FUNCTION "Axis_Control" : VOID	// FC 38
TITLE = Axis control
//KNOW_HOW_PROTECT
//
VERSION : 0.1
VAR_INPUT
  Enable : BOOL ;
  Axis_Enc_Num : BYTE ;
  Axis_Plus_LimitSwitch : BOOL ;
  Axis_Minus_LimitSwitch : BOOL ;
  Axis_Ref_Switch : BOOL ;
  Axis_PositContr : BOOL ;
  Run_Mode : BOOL ;
  Axis_1st_Ref_Active : BOOL ;
  Axis_2nd_Ref_Active : BOOL ;
  Axis_Limitactive : DWORD ;
END_VAR
VAR_OUTPUT
  Axis_PulseEnable : BOOL ;
  Axis_ContrEnable : BOOL ;
  Axis_PosMeas1 : BOOL ;
  Axis_PosMeas2 : BOOL ;
  Axis_ORactive : BOOL ;
  Axis_Refactive : BOOL ;
  Axis_BreakActive : BOOL ;
  Axis_Plus_Limit : BOOL ;
  Axis_Minus_Limit : BOOL ;
  Axis_refpoint : BOOL ;
END_VAR
BEGIN
NETWORK
TITLE =
      L     1;
      L     #Axis_Enc_Num;
      -I;
      JN    M001;
      A     "ONE";
      =     #Axis_PosMeas1;
      AN    #Axis_PosMeas1;
      =     #Axis_PosMeas2;
      JU    M002;
M001: A     "ONE";
      =     #Axis_PosMeas2;
      AN    #Axis_PosMeas2;
      =     #Axis_PosMeas1;
M002: A     #Enable;
      =     #Axis_PulseEnable;
      =     #Axis_ContrEnable;
      AN    #Run_Mode;
      =     #Axis_ORactive;
      A     #Axis_PositContr;
      =     #Axis_BreakActive;
      A     #Axis_1st_Ref_Active;
      O     #Axis_2nd_Ref_Active;
      =     #Axis_Refactive;
      A     #Axis_Ref_Switch;
      =     #Axis_refpoint;
      L     #Axis_Limitactive;
      L     1.000000e+00;
      -R;
      JZ    NONE;
      AN    #Axis_Plus_LimitSwitch;
      =     #Axis_Plus_Limit;
      AN    #Axis_Minus_LimitSwitch;
      =     #Axis_Minus_Limit;
      JU    EXIT;
NONE: A     "Reset_Key";
      R     #Axis_Plus_Limit;
      R     #Axis_Minus_Limit;
EXIT: BE;
END_FUNCTION

FUNCTION "System_Date" : VOID	// FC 39
TITLE = function
//KNOW_HOW_PROTECT 
//M153.6,MW316 DB110,DB120,DB125
//
VERSION : 0.1
BEGIN
NETWORK
TITLE =
//ReadSysTime M153.6,MW316 DB110,DB120,DB125
      CALL  "READ_CLK" (
           RET_VAL                  := MW 316,
           CDT                      := P#DB110.DBX 0.0);
      L     DB110.DBB 0;	//YEAR
      BTI;
      T     DB125.DBB 0;
      T     "USER_DB5".STAT0[5];
      L     DB110.DBB 1;	//MONTH
      BTI;
      T     DB125.DBB 1;
      T     "USER_DB5".STAT0[6];
      L     DB110.DBB 2;	//DAY
      BTI;
      T     DB125.DBB 2;
      T     "USER_DB5".STAT0[7];
      L     DB110.DBB 3;	//HOUR
      BTI;
      T     DB125.DBB 3;
      T     "USER_DB5".STAT0[8];
      L     DB110.DBB 4;	//MINUTE
      BTI;
      T     DB125.DBB 4;
      T     "USER_DB5".STAT0[9];
      L     DB110.DBB 5;	//SECOND
      BTI;
      T     DB125.DBB 5;
      T     "USER_DB5".STAT0[10];
      A     "Time_Lock_Active";
      JC    EXIT;
      L     DB120.DBD 70;
      L     1.000000e+00;
      -R;
      JN    ZERO;
      L     "USER_DB5".STAT0[5];	//YEAR
      L     10000;
      *I;
      T     DB125.DBD 30;
      L     "USER_DB5".STAT0[6];	//MONTH
      L     100;
      *I;
      T     DB125.DBD 40;
      L     "USER_DB5".STAT0[7];	//DATE
      T     DB125.DBD 50;
      L     DB125.DBD 30;
      +D;
      T     DB125.DBD 60;
      L     DB125.DBD 40;
      +D;
      T     DB125.DBD 70;
      L     DB120.DBD 80;
      RND;
      T     DB125.DBD 80;
      L     DB125.DBD 70;
      L     DB125.DBD 80;
      >=I;
      JC    ONE;
      JU    ZERO;
EXIT: L     DB120.DBD 70;
      L     1.000000e+00;
      -R;
      JZ    ONE;
      A     "Reset_Key";
      A     "Auto_Key";
      A     "MDA_Key";
      R     "Time_Lock_Active";
      JU    END;
ONE:  S     "Time_Lock_Active";
      JU    END;
ZERO: R     "Time_Lock_Active";
END:  BE;
END_FUNCTION

FUNCTION "X_BACK_Control" : VOID	// FC 40
TITLE = X_BACK
//M155.0_M155.7,MW322,MW324,DB16,DB106,DB159,FB4,FC9,T27
//KNOW_HOW_PROTECT
//
VERSION : 0.1
BEGIN
NETWORK
TITLE = M155.0_M155.7,MW322,MW324,DB16,DB106,DB159,FB4,FC9,T27
      A     "Auto_LED";
      L     S5T#500MS;
      SD    "KT17";
      A     "KT17";
      =     M 155.0;
      A     "Reset_Key";
      A     M 155.1;
      R     M 155.0;
      R     M 155.1;
      CALL  "PI_SERV" , DB 159 (
           DIX 0.0                  := M 155.0,
           DIW 2                    := W#16#1002,
           DIW 4                    := 26,
           DIW 6                    := 16,
           DID 8                    := P#DBX 18.0,
           DIW 12                   := 1,
           DIW 14                   := W#16#1002,
           DIW 16                   := 34,
           DIW 18                   := 106,
           DID 20                   := P#DBX 34.0,
           DIW 24                   := W#16#1002,
           DIW 26                   := 34,
           DIW 28                   := 106,
           DID 30                   := P#DBX 0.0,
           DIW 54                   := 1,
           DIW 56                   := 1,
           DIX 74.0                 := M 155.1,
           DIX 74.1                 := M 155.2,
           DIW 76                   := MW 322);
      A(;
      O     DB11.DBX 6.0;
      O     DB11.DBX 6.1;
      );
      A     DB21.DBX 35.0;
      AN    DB21.DBX 197.6;
      AN    "Reset_Key";
      =     M 156.0;
      CALL  "Single Key control" (
           CH1_M_ON                 := DB21.DBX 201.0,
           CH2_M_ON                 := FALSE,
           CH1_M_OFF                := DB21.DBX 201.1,
           CH2_M_OFF                := FALSE,
           Key                      := "T13_X轴快退",
           Var1                     := M 156.1,
           Var2                     := M 156.2,
           Var3_up                  := FALSE,
           Protect                  := M 156.0,
           KeyEnableMode            := TRUE,
           KA                       := M 156.3,
           LED                      := M 156.3);
      A(;
      O     DB2.DBX 181.4;
      O     DB2.DBX 181.7;
      O     DB2.DBX 182.0;
      O     DB2.DBX 182.5;
      O     DB2.DBX 183.1;
      O     DB2.DBX 183.2;
      O     DB2.DBX 183.5;
      );
      A     M 156.0;
      AN    DB21.DBX 201.1;
      =     M 156.4;
      A(;
      O     DB2.DBX 181.5;
      O     DB2.DBX 182.6;
      );
      A     M 156.0;
      AN    DB21.DBX 201.1;
      =     M 156.5;
      A     M 156.0;
      A     "-UPS_电池供电";
      =     M 156.6;
      A     M 156.3;
      =     DB10.DBX 1.1;
      O     M 156.4;
      O     M 156.5;
      O     M 156.6;
      =     DB10.DBX 125.5;
      O     M 156.3;
      O     M 156.4;
      O     M 156.5;
      O     M 156.6;
      =     "T13_LED_X轴快退";
      A     "T13_LED_X轴快退";
//   A     "NC".A_Set_Inp2
//    L     S5T#100MS
//    SD    "T_ASUP_DELAY1"
//    AN    "NC".A_Set_Inp2
//    L     S5T#1S
//     SF    "T_ASUP_DELAY2"
//     A     "T_ASUP_DELAY1"
//     A     "T_ASUP_DELAY2"
//     =     "NC".A_Set_Inp19
//     A     "NC".A_Set_Inp2
//      L     S5T#600MS
//      SD    "T_ASUP_DELAY3"
//      O     M    156.4
//      O     M    156.5
//      =     "NC".A_Set_Inp22
//      A     "T_ASUP_DELAY3"
      A     M 155.2;
      =     M 155.3;
      A     "Reset_Key";
      A(;
      O     M 155.6;
      O     M 155.7;
      );
      R     M 155.3;
      R     M 155.6;
      R     M 155.7;
      CALL  "ASUP" (
           $1                       := M 155.3,
           $2                       := 1,
           $3                       := 1,
           $4                       := M 155.4,
           $5                       := M 155.5,
           $6                       := M 155.6,
           $7                       := M 155.7,
           $8                       := P#M 324.0);
      A     M 155.6;
      =     DB2.DBX 183.7;
      BE;
END_FUNCTION

FUNCTION "Grinding_Speed_2" : VOID	// FC 41
//M157.0__M157.7 MW328,DB126,DB153
VERSION : 0.1
BEGIN
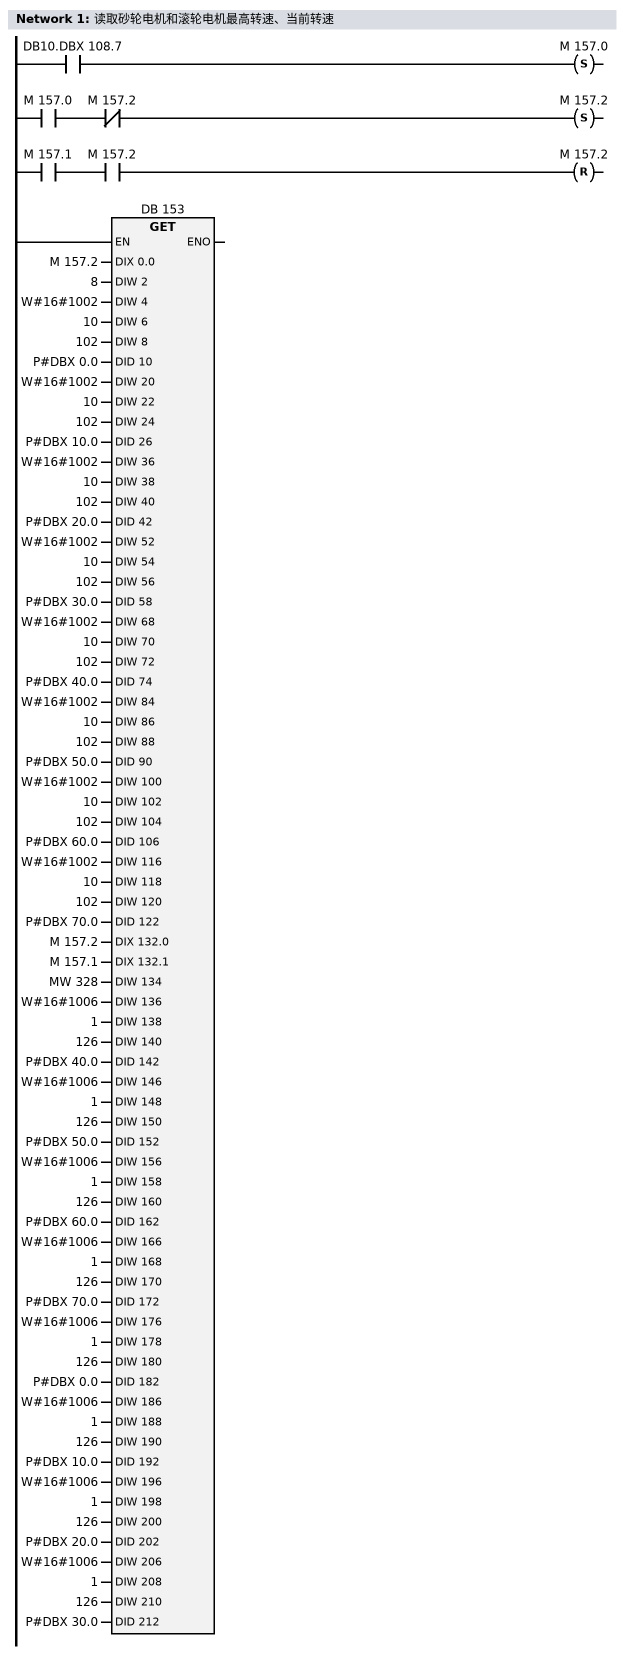
NETWORK
TITLE = 读取砂轮电机和滚轮电机最高转速、当前转速
      A     DB10.DBX 108.7;
      S     M 157.0;
      A     M 157.0;
      AN    M 157.2;
      S     M 157.2;
      A     M 157.1;
      A     M 157.2;
      R     M 157.2;
      CALL  "GET" , DB 153 (
           DIX 0.0                  := M 157.2,
           DIW 2                    := 8,
           DIW 4                    := W#16#1002,
           DIW 6                    := 10,
           DIW 8                    := 102,
           DID 10                   := P#DBX 0.0,
           DIW 20                   := W#16#1002,
           DIW 22                   := 10,
           DIW 24                   := 102,
           DID 26                   := P#DBX 10.0,
           DIW 36                   := W#16#1002,
           DIW 38                   := 10,
           DIW 40                   := 102,
           DID 42                   := P#DBX 20.0,
           DIW 52                   := W#16#1002,
           DIW 54                   := 10,
           DIW 56                   := 102,
           DID 58                   := P#DBX 30.0,
           DIW 68                   := W#16#1002,
           DIW 70                   := 10,
           DIW 72                   := 102,
           DID 74                   := P#DBX 40.0,
           DIW 84                   := W#16#1002,
           DIW 86                   := 10,
           DIW 88                   := 102,
           DID 90                   := P#DBX 50.0,
           DIW 100                  := W#16#1002,
           DIW 102                  := 10,
           DIW 104                  := 102,
           DID 106                  := P#DBX 60.0,
           DIW 116                  := W#16#1002,
           DIW 118                  := 10,
           DIW 120                  := 102,
           DID 122                  := P#DBX 70.0,
           DIX 132.0                := M 157.2,
           DIX 132.1                := M 157.1,
           DIW 134                  := MW 328,
           DIW 136                  := W#16#1006,
           DIW 138                  := 1,
           DIW 140                  := 126,
           DID 142                  := P#DBX 40.0,
           DIW 146                  := W#16#1006,
           DIW 148                  := 1,
           DIW 150                  := 126,
           DID 152                  := P#DBX 50.0,
           DIW 156                  := W#16#1006,
           DIW 158                  := 1,
           DIW 160                  := 126,
           DID 162                  := P#DBX 60.0,
           DIW 166                  := W#16#1006,
           DIW 168                  := 1,
           DIW 170                  := 126,
           DID 172                  := P#DBX 70.0,
           DIW 176                  := W#16#1006,
           DIW 178                  := 1,
           DIW 180                  := 126,
           DID 182                  := P#DBX 0.0,
           DIW 186                  := W#16#1006,
           DIW 188                  := 1,
           DIW 190                  := 126,
           DID 192                  := P#DBX 10.0,
           DIW 196                  := W#16#1006,
           DIW 198                  := 1,
           DIW 200                  := 126,
           DID 202                  := P#DBX 20.0,
           DIW 206                  := W#16#1006,
           DIW 208                  := 1,
           DIW 210                  := 126,
           DID 212                  := P#DBX 30.0);	//R296:备用1 / R297:滚轮电机转速 / R298:备用2 / R299:砂轮电机转速 / R500:备用1上限 / R501:滚轮电机最高转速 / R502:备用2上限 / R503:砂轮电机最高转速
NETWORK
TITLE = 速度计算
      L     DB126.DBD 70;	//砂轮电机当前转速
      L     DB126.DBD 30;	//砂轮电机最高转速
      -R;
      JP    SPE0;
      L     DB126.DBD 70;
      T     DB126.DBD 80;	//砂轮电机实际转速
      JU    SPE1;
SPE0: L     DB126.DBD 30;
      T     DB126.DBD 80;
SPE1: L     DB126.DBD 50;	//滚轮电机当前转速
      L     DB126.DBD 10;	//滚轮电机最高转速
      -R;
      JP    SPE2;
      L     DB126.DBD 50;
      T     DB126.DBD 90;	//滚轮电机实际转速
      JU    SPE3;
SPE2: L     DB126.DBD 10;
      T     DB126.DBD 90;
NETWORK
TITLE = 模拟电压计算输出
//砂轮模拟电压输出计算
SPE3: L     1.020000e+02;
      L     DB126.DBD 30;
      /R;
      T     DB126.DBD 100;
      L     DB126.DBD 80;
      L     DB126.DBD 100;
      *R;
      T     DB126.DBD 110;
      TRUNC;
      T     DB126.DBD 120;
//滚轮模拟电压输出计算
      L     1.020000e+02;
      L     DB126.DBD 10;
      /R;
      T     DB126.DBD 130;
      L     DB126.DBD 90;
      L     DB126.DBD 130;
      *R;
      T     DB126.DBD 140;
      L     DB126.DBD 140;
      TRUNC;
      T     DB126.DBD 150;
//模拟电压输出
      L     B#16#55;
      T     QB 56;
      L     B#16#1;
      T     QB 57;
      L     "USER_DB6".STAT0[61];
      L     102;
      >=I;
      =     M 157.3;
      L     0;
      L     "USER_DB6".STAT0[61];
      >=I;
      =     M 157.4;
      A     "ONE";
      A     M 157.3;
      JC    SPP1;
      A     "ONE";
      A     M 157.4;
      JC    SPP2;
      L     "USER_DB6".STAT0[61];
      T     "USER_DB6".STAT0[81];
      JU    SPP3;
SPP1: L     102;
      T     "USER_DB6".STAT0[81];
      JU    SPP3;
SPP2: L     0;
      T     "USER_DB6".STAT0[81];
SPP3: L     "USER_DB6".STAT0[81];
      T     QW 60;	//模拟电压1输出
      L     "USER_DB6".STAT0[76];
      L     102;
      >=I;
      =     M 157.5;
      L     0;
      L     "USER_DB6".STAT0[76];
      >=I;
      =     M 157.6;
      A     "ONE";
      A     M 157.5;
      JC    SPP4;
      A     "ONE";
      A     M 157.6;
      JC    SPP5;
      L     "USER_DB6".STAT0[76];
      T     "USER_DB6".STAT0[86];
      JU    SPP6;
SPP4: L     102;
      T     "USER_DB6".STAT0[86];
      JU    SPP6;
SPP5: L     0;
      T     "USER_DB6".STAT0[86];
SPP6: L     "USER_DB6".STAT0[86];
      T     QW 62;	//模拟电压2输出 
      A     "Reset_Key";
      R     M 157.2;
      BE;
END_FUNCTION

FUNCTION "Truss manipulator" : VOID	// FC 42
TITLE = 桁架机械手臂控制
//MW20
VERSION : 0.1
VAR_INPUT
  IN0 : BOOL ;	//取成品到位
  IN1 : BOOL ;	//送毛坯到位
  IN2 : BOOL ;	//手爪收回到位
  IN3 : BOOL ;	//备用接收信号1
  IN4 : BOOL ;	//备用接收信号2
END_VAR
VAR_OUTPUT
  OUT0 : BOOL ;	//罩壳门打开信号
  OUT1 : BOOL ;	//预完成信号
  OUT2 : BOOL ;	//机床故障信号
  OUT3 : BOOL ;	//卡盘松开完成信号
  OUT4 : BOOL ;	//卡盘夹紧完成信号
  OUT5 : BOOL ;	//备用输出1
  OUT6 : BOOL ;	//备用输出2
  OUT7 : BOOL ;	//备用输出3
END_VAR
BEGIN
NETWORK
TITLE = Set digi. NCK input 30、31、32、33、34
      A     #IN0;
      =     DB10.DBX 127.5;
      A     #IN1;
      =     DB10.DBX 127.6;
      A     #IN2;
      =     DB10.DBX 127.7;
      A     #IN3;
      =     DB10.DBX 129.0;
      A     #IN4;
      =     DB10.DBX 129.1;
NETWORK
TITLE = Set digi. NCK input 36、37、38、39、40  MW20
      A     "ONE";
      =     L 0.0;
      A     L 0.0;
      A     DB21.DBX 204.0;
      FP    M 20.0;
      S     DB10.DBX 129.3;
      A     L 0.0;
      A(;
      O     "Reset_Key";
      O     M 16.2;
      O     DB21.DBX 204.1;
      );
      FP    M 20.1;
      R     DB10.DBX 129.3;
      A     L 0.0;
      A     DB21.DBX 204.2;
      FP    M 20.2;
      S     DB10.DBX 129.4;
      A     L 0.0;
      A(;
      O     "Reset_Key";
      O     M 16.2;
      O     DB21.DBX 204.3;
      );
      FP    M 20.3;
      R     DB10.DBX 129.4;
      A     L 0.0;
      A     DB21.DBX 204.4;
      FP    M 20.4;
      S     DB10.DBX 129.5;
      A     L 0.0;
      A(;
      O     "Reset_Key";
      O     M 16.2;
      O     DB21.DBX 204.5;
      );
      FP    M 20.5;
      R     DB10.DBX 129.5;
      A     L 0.0;
      A     DB21.DBX 204.6;
      FP    M 20.6;
      S     DB10.DBX 129.6;
      A     L 0.0;
      A(;
      O     "Reset_Key";
      O     M 16.2;
      O     DB21.DBX 204.7;
      );
      FP    M 20.7;
      R     DB10.DBX 129.6;
      A     L 0.0;
      A     DB21.DBX 205.0;
      FP    M 21.0;
      S     DB10.DBX 129.7;
      A     L 0.0;
      A(;
      O     "Reset_Key";
      O     M 16.2;
      O     DB21.DBX 205.1;
      );
      FP    M 21.1;
      R     DB10.DBX 129.7;
      A     L 0.0;
      A(;
      ON    "-SB0_急停按钮";
      ON    "-SB1_辅助急停1";
      ON    "-SB2_辅助急停2";
      );
      =     "EMG_Active";
      A     L 0.0;
      A(;
      O     DB21.DBX 35.1;
      O     DB21.DBX 35.2;
      );
      =     "Chan1_Stop";
NETWORK
TITLE = NC给机械手信号
      A     DB10.DBX 129.3;
      =     #OUT0;
      A     DB10.DBX 129.4;
      =     #OUT1;
      A     DB10.DBX 129.5;
      =     #OUT2;
      A     DB10.DBX 129.6;
      =     #OUT3;
      A     DB10.DBX 129.7;
      =     #OUT4;
      BE;
END_FUNCTION

// FC 1005: know-how protected block, not included

// FC 1006: know-how protected block, not included

DATA_BLOCK DB 4
AUTHOR : NUMERIK
FAMILY : _800D
NAME : Basics
VERSION : 4.5
  STRUCT
   BOfeld0 : WORD  := W#16#CD54;	//Channel 1-8 ever 18 Bits
   BOfeld2 : WORD  := W#16#3553;
   BOfeld4 : WORD  := W#16#D54C;
   BOfeld6 : WORD  := W#16#5533;
   BOfeld8 : WORD  := W#16#55CD;
   BOfeld10 : WORD  := W#16#5435;
   BOfeld12 : WORD  := W#16#53D5;
   BOfeld14 : WORD  := W#16#4C55;
   BOfeld16 : WORD  := W#16#3355;
   BOfeld18 : WORD  := W#16#5555;	//18 Axes/Spindles ever 2 Bit
   BOfeld20 : WORD  := W#16#5555;
   BOfeld22 : WORD  := W#16#F5F0;	//10 User data area ever 8 Bit (Begin: DBB23)
   BOfeld24 : WORD  := W#16#F0F0;
   BOfeld26 : WORD  := W#16#F0F0;
   BOfeld28 : WORD  := W#16#F0F0;
   BOfeld30 : WORD  := W#16#F0F0;
   BOfeld32 : WORD  := W#16#F0F0;
   BOfeld34 : WORD  := W#16#F0F0;
   BOfeld36 : WORD  := W#16#F0F0;
   BOfeld38 : WORD  := W#16#F0F0;
   BOfeld40 : WORD  := W#16#F0F0;
   BOfeld42 : WORD  := W#16#F0F0;
   BOfeld44 : WORD  := W#16#F0F0;
   BOfeld46 : WORD  := W#16#F0F0;
   BOfeld48 : WORD  := W#16#F0F0;
   BOfeld50 : WORD  := W#16#F0F0;
   BOfeld52 : WORD  := W#16#F0F0;
   BOfeld54 : WORD  := W#16#F0F0;
   BOfeld56 : WORD  := W#16#F0F0;
   BOfeld58 : WORD  := W#16#F0F0;
   BOfeld60 : WORD  := W#16#F0F0;
   BOfeld62 : BYTE  := B#16#F0;
   NumUser : BYTE  := B#16#A;
   maganz : BYTE ;	//for TM, number of Magazine
   wzv : BYTE ;
   wzvdat : ARRAY  [1 .. 160 ] OF BYTE ;	//32 Magazine, possibly ever 5 Byte + Spindle
  END_STRUCT ;	
BEGIN
   BOfeld0 := W#16#CD54;
   BOfeld2 := W#16#3553;
   BOfeld4 := W#16#D54C;
   BOfeld6 := W#16#5533;
   BOfeld8 := W#16#55CD;
   BOfeld10 := W#16#5435;
   BOfeld12 := W#16#53D5;
   BOfeld14 := W#16#4C55;
   BOfeld16 := W#16#3355;
   BOfeld18 := W#16#5555;
   BOfeld20 := W#16#5555;
   BOfeld22 := W#16#F5F0;
   BOfeld24 := W#16#F0F0;
   BOfeld26 := W#16#F0F0;
   BOfeld28 := W#16#F0F0;
   BOfeld30 := W#16#F0F0;
   BOfeld32 := W#16#F0F0;
   BOfeld34 := W#16#F0F0;
   BOfeld36 := W#16#F0F0;
   BOfeld38 := W#16#F0F0;
   BOfeld40 := W#16#F0F0;
   BOfeld42 := W#16#F0F0;
   BOfeld44 := W#16#F0F0;
   BOfeld46 := W#16#F0F0;
   BOfeld48 := W#16#F0F0;
   BOfeld50 := W#16#F0F0;
   BOfeld52 := W#16#F0F0;
   BOfeld54 := W#16#F0F0;
   BOfeld56 := W#16#F0F0;
   BOfeld58 := W#16#F0F0;
   BOfeld60 := W#16#F0F0;
   BOfeld62 := B#16#F0;
   NumUser := B#16#A;
END_DATA_BLOCK

DATA_BLOCK DB 5
AUTHOR : NUMERIK
FAMILY : _800D
NAME : Basics
VERSION : 4.5
  STRUCT
   Ch1_DB2_310 : BOOL  := TRUE;	// (Channel 1-10 ever 18 Bits):  error message
   Ch1_DB2_311 : BOOL ;	// Channel 1, DB2.DBB311; operational message
   Ch1_DB2_312 : BOOL  := TRUE;	// Channel 1, DB2.DBB312; error message
   Ch1_DB2_313 : BOOL  := TRUE;	// error message
   Ch1_DB2_314 : BOOL ;	// operational message
   Ch1_DB2_315 : BOOL ;	// operational message
   Ch1_DB2_316 : BOOL  := TRUE;	// error message
   Ch1_DB2_317 : BOOL  := TRUE;	// error message
   Ch1_DB2_318 : BOOL ;	// operational message
   Ch1_DB2_319 : BOOL ;	// operational message
   Ch1_DB2_320 : BOOL  := TRUE;	// error message
   Ch1_DB2_321 : BOOL ;	// operational message
   Ch1_DB2_322 : BOOL  := TRUE;	// error message
   Ch1_DB2_323 : BOOL ;	// operational message
   Ch1_DB2_324 : BOOL  := TRUE;	// error message
   Ch1_DB2_325 : BOOL ;	// operational message
   Ch1_DB2_326 : BOOL  := TRUE;	// error message
   Ch1_DB2_327 : BOOL ;	// operational message
   Ch2_DB2_328 : BOOL  := TRUE;	// Channel 2, DB2.DBB328; error message
   Ch2_DB2_329 : BOOL ;	// Channel 2, DB2.DBB329; operational message
   Ch2_DB2_330 : BOOL  := TRUE;	// error message
   Ch2_DB2_331 : BOOL  := TRUE;	// error message
   Ch2_DB2_332 : BOOL ;	// operational message
   Ch2_DB2_333 : BOOL ;	// operational message
   Ch2_DB2_334 : BOOL  := TRUE;	// error message
   Ch2_DB2_335 : BOOL  := TRUE;	// error message
   Ch2_DB2_336 : BOOL ;	// operational message
   Ch2_DB2_337 : BOOL ;	// operational message
   Ch2_DB2_338 : BOOL  := TRUE;	// error message
   Ch2_DB2_339 : BOOL ;	// operational message
   Ch2_DB2_340 : BOOL  := TRUE;	// error message
   Ch2_DB2_341 : BOOL ;	// operational message
   Ch2_DB2_342 : BOOL  := TRUE;	// error message
   Ch2_DB2_343 : BOOL ;	// operational message
   Ch2_DB2_344 : BOOL  := TRUE;	// error message
   Ch2_DB2_345 : BOOL ;	// operational message
   Ch3_DB2_346 : BOOL  := TRUE;	// Channel 3, DB2.DBB346; error message
   Ch3_DB2_347 : BOOL ;	// Channel 3, DB2.DBB347; operational message
   Ch3_DB2_348 : BOOL  := TRUE;	// error message
   Ch3_DB2_349 : BOOL  := TRUE;	// error message
   Ch3_DB2_350 : BOOL ;	// operational message
   Ch3_DB2_351 : BOOL ;	// operational message
   Ch3_DB2_352 : BOOL  := TRUE;	// error message
   Ch3_DB2_353 : BOOL  := TRUE;	// error message
   Ch3_DB2_354 : BOOL ;	// operational message
   Ch3_DB2_355 : BOOL ;	// operational message
   Ch3_DB2_356 : BOOL  := TRUE;	// error message
   Ch3_DB2_357 : BOOL ;	// operational message
   Ch3_DB2_358 : BOOL  := TRUE;	// error message
   Ch3_DB2_359 : BOOL ;	// operational message
   Ch3_DB2_360 : BOOL  := TRUE;	// error message
   Ch3_DB2_361 : BOOL ;	// operational message
   Ch3_DB2_362 : BOOL  := TRUE;	// error message
   Ch3_DB2_363 : BOOL ;	// operational message
   Ch4_DB2_364 : BOOL  := TRUE;	// Channel 4, DB2.DBB364; error message
   Ch4_DB2_365 : BOOL ;	// Channel 4, DB2.DBB365; operational message
   Ch4_DB2_366 : BOOL  := TRUE;	// error message
   Ch4_DB2_367 : BOOL  := TRUE;	// error message
   Ch4_DB2_368 : BOOL ;	// operational message
   Ch4_DB2_369 : BOOL ;	// operational message
   Ch4_DB2_370 : BOOL  := TRUE;	// error message
   Ch4_DB2_371 : BOOL  := TRUE;	// error message
   Ch4_DB2_372 : BOOL ;	// operational message
   Ch4_DB2_373 : BOOL ;	// operational message
   Ch4_DB2_374 : BOOL  := TRUE;	// error message
   Ch4_DB2_375 : BOOL ;	// operational message
   Ch4_DB2_376 : BOOL  := TRUE;	// error message
   Ch4_DB2_377 : BOOL ;	// operational message
   Ch4_DB2_378 : BOOL  := TRUE;	// error message
   Ch4_DB2_379 : BOOL ;	// operational message
   Ch4_DB2_380 : BOOL  := TRUE;	// error message
   Ch4_DB2_381 : BOOL ;	// operational message
   Ch5_DB2_382 : BOOL  := TRUE;	// Channel 5, DB2.DBB382; error message
   Ch5_DB2_383 : BOOL ;	// Channel 5, DB2.DBB383; operational message
   Ch5_DB2_384 : BOOL  := TRUE;	// error message
   Ch5_DB2_385 : BOOL  := TRUE;	// error message
   Ch5_DB2_386 : BOOL ;	// operational message
   Ch5_DB2_387 : BOOL ;	// operational message
   Ch5_DB2_388 : BOOL  := TRUE;	// error message
   Ch5_DB2_389 : BOOL  := TRUE;	// error message
   Ch5_DB2_390 : BOOL ;	// operational message
   Ch5_DB2_391 : BOOL ;	// operational message
   Ch5_DB2_392 : BOOL  := TRUE;	// error message
   Ch5_DB2_393 : BOOL ;	// operational message
   Ch5_DB2_394 : BOOL  := TRUE;	// error message
   Ch5_DB2_395 : BOOL ;	// operational message
   Ch5_DB2_396 : BOOL  := TRUE;	// error message
   Ch5_DB2_397 : BOOL ;	// operational message
   Ch5_DB2_398 : BOOL  := TRUE;	// error message
   Ch5_DB2_399 : BOOL ;	// operational message
   Ch6_DB2_400 : BOOL  := TRUE;	// Channel 6, DB2.DBB400; error message
   Ch6_DB2_401 : BOOL ;	// Channel 6, DB2.DBB401; operational message
   Ch6_DB2_402 : BOOL  := TRUE;	// error message
   Ch6_DB2_403 : BOOL  := TRUE;	// error message
   Ch6_DB2_404 : BOOL ;	// operational message
   Ch6_DB2_405 : BOOL ;	// operational message
   Ch6_DB2_406 : BOOL  := TRUE;	// error message
   Ch6_DB2_407 : BOOL  := TRUE;	// error message
   Ch6_DB2_408 : BOOL ;	// operational message
   Ch6_DB2_409 : BOOL ;	// operational message
   Ch6_DB2_410 : BOOL  := TRUE;	// error message
   Ch6_DB2_411 : BOOL ;	// operational message
   Ch6_DB2_412 : BOOL  := TRUE;	// error message
   Ch6_DB2_413 : BOOL ;	// operational message
   Ch6_DB2_414 : BOOL  := TRUE;	// error message
   Ch6_DB2_415 : BOOL ;	// operational message
   Ch6_DB2_416 : BOOL  := TRUE;	// error message
   Ch6_DB2_417 : BOOL ;	// operational message
   Ch7_DB2_418 : BOOL  := TRUE;	// Channel 7, DB2.DBB418; error message
   Ch7_DB2_419 : BOOL ;	// Channel 7, DB2.DBB419; operational message
   Ch7_DB2_420 : BOOL  := TRUE;	// error message
   Ch7_DB2_421 : BOOL  := TRUE;	// error message
   Ch7_DB2_422 : BOOL ;	// operational message
   Ch7_DB2_423 : BOOL ;	// operational message
   Ch7_DB2_424 : BOOL  := TRUE;	// error message
   Ch7_DB2_425 : BOOL  := TRUE;	// error message
   Ch7_DB2_426 : BOOL ;	// operational message
   Ch7_DB2_427 : BOOL ;	// operational message
   Ch7_DB2_428 : BOOL  := TRUE;	// error message
   Ch7_DB2_429 : BOOL ;	// operational message
   Ch7_DB2_430 : BOOL  := TRUE;	// error message
   Ch7_DB2_431 : BOOL ;	// operational message
   Ch7_DB2_432 : BOOL  := TRUE;	// error message
   Ch7_DB2_433 : BOOL ;	// operational message
   Ch7_DB2_434 : BOOL  := TRUE;	// error message
   Ch7_DB2_435 : BOOL ;	// operational message
   Ch8_DB2_436 : BOOL  := TRUE;	// Channel 8, DB2.DBB436; error message
   Ch8_DB2_437 : BOOL ;	// Channel 8, DB2.DBB437; operational message
   Ch8_DB2_438 : BOOL  := TRUE;	// error message
   Ch8_DB2_439 : BOOL  := TRUE;	// error message
   Ch8_DB2_440 : BOOL ;	// operational message
   Ch8_DB2_441 : BOOL ;	// operational message
   Ch8_DB2_442 : BOOL  := TRUE;	// error message
   Ch8_DB2_443 : BOOL  := TRUE;	// error message
   Ch8_DB2_444 : BOOL ;	// operational message
   Ch8_DB2_445 : BOOL ;	// operational message
   Ch8_DB2_446 : BOOL  := TRUE;	// error message
   Ch8_DB2_447 : BOOL ;	// operational message
   Ch8_DB2_448 : BOOL  := TRUE;	// error message
   Ch8_DB2_449 : BOOL ;	// operational message
   Ch8_DB2_450 : BOOL  := TRUE;	// error message
   Ch8_DB2_451 : BOOL ;	// operational message
   Ch8_DB2_452 : BOOL  := TRUE;	// error message
   Ch8_DB2_453 : BOOL ;	// operational message
   Ch9_DB2_454 : BOOL  := TRUE;	// Channel 9, DB2.DBB454; error message
   Ch9_DB2_455 : BOOL ;	// Channel 9, DB2.DBB455; operational message
   Ch9_DB2_456 : BOOL  := TRUE;	// error message
   Ch9_DB2_457 : BOOL  := TRUE;	// error message
   Ch9_DB2_458 : BOOL ;	// operational message
   Ch9_DB2_459 : BOOL ;	// operational message
   Ch9_DB2_460 : BOOL  := TRUE;	// error message
   Ch9_DB2_461 : BOOL  := TRUE;	// error message
   Ch9_DB2_462 : BOOL ;	// operational message
   Ch9_DB2_463 : BOOL ;	// operational message
   Ch9_DB2_464 : BOOL  := TRUE;	// error message
   Ch9_DB2_465 : BOOL ;	// operational message
   Ch9_DB2_466 : BOOL  := TRUE;	// error message
   Ch9_DB2_467 : BOOL ;	// operational message
   Ch9_DB2_468 : BOOL  := TRUE;	// error message
   Ch9_DB2_469 : BOOL ;	// operational message
   Ch9_DB2_470 : BOOL  := TRUE;	// error message
   Ch9_DB2_471 : BOOL ;	// operational message
   Ch10_DB2_472 : BOOL  := TRUE;	// Channel 10, DB2.DBB472; error message
   Ch10_DB2_473 : BOOL ;	// Channel 10, DB2.DBB473; operational message
   Ch10_DB2_474 : BOOL  := TRUE;	// error message
   Ch10_DB2_475 : BOOL  := TRUE;	// error message
   Ch10_DB2_476 : BOOL ;	// operational message
   Ch10_DB2_477 : BOOL ;	// operational message
   Ch10_DB2_478 : BOOL  := TRUE;	// error message
   Ch10_DB2_479 : BOOL  := TRUE;	// error message
   Ch10_DB2_480 : BOOL ;	// operational message
   Ch10_DB2_481 : BOOL ;	// operational message
   Ch10_DB2_482 : BOOL  := TRUE;	// error message
   Ch10_DB2_483 : BOOL ;	// operational message
   Ch10_DB2_484 : BOOL  := TRUE;	// error message
   Ch10_DB2_485 : BOOL ;	// operational message
   Ch10_DB2_486 : BOOL  := TRUE;	// error message
   Ch10_DB2_487 : BOOL ;	// operational message
   Ch10_DB2_488 : BOOL  := TRUE;	// error message
   Ch10_DB2_489 : BOOL ;	// operational message
   Ax1_DB2_490 : BOOL  := TRUE;	// (32 Axes/Spindles ever 2 Bit):  error message
   Ax1_DB2_491 : BOOL ;	// Axis 1, DB2.DBB491; operational message
   Ax2_DB2_492 : BOOL  := TRUE;	// Axis 2, DB2.DBB492; error message
   Ax2_DB2_493 : BOOL ;	// Axis 2, DB2.DBB493; operational message
   Ax3_DB2_494 : BOOL  := TRUE;	// error message
   Ax3_DB2_495 : BOOL ;	// operational message
   Ax4_DB2_496 : BOOL  := TRUE;	// error message
   Ax4_DB2_497 : BOOL ;	// operational message
   Ax5_DB2_498 : BOOL  := TRUE;	// error message
   Ax5_DB2_499 : BOOL ;	// operational message
   Ax6_DB2_500 : BOOL  := TRUE;	// error message
   Ax6_DB2_501 : BOOL ;	// operational message
   Ax7_DB2_502 : BOOL  := TRUE;	// error message
   Ax7_DB2_503 : BOOL ;	// operational message
   Ax8_DB2_504 : BOOL  := TRUE;	// error message
   Ax8_DB2_505 : BOOL ;	// operational message
   Ax9_DB2_506 : BOOL  := TRUE;	// error message
   Ax9_DB2_507 : BOOL ;	// operational message
   Ax10_DB2_508 : BOOL  := TRUE;	// error message
   Ax10_DB2_509 : BOOL ;	// operational message
   Ax11_DB2_510 : BOOL  := TRUE;	// error message
   Ax11_DB2_511 : BOOL ;	// operational message
   Ax12_DB2_512 : BOOL  := TRUE;	// error message
   Ax12_DB2_513 : BOOL ;	// operational message
   Ax13_DB2_514 : BOOL  := TRUE;	// error message
   Ax13_DB2_515 : BOOL ;	// operational message
   Ax14_DB2_516 : BOOL  := TRUE;	// error message
   Ax14_DB2_517 : BOOL ;	// operational message
   Ax15_DB2_518 : BOOL  := TRUE;	// error message
   Ax15_DB2_519 : BOOL ;	// operational message
   Ax16_DB2_520 : BOOL  := TRUE;	// error message
   Ax16_DB2_521 : BOOL ;	// operational message
   Ax17_DB2_522 : BOOL  := TRUE;	// error message
   Ax17_DB2_523 : BOOL ;	// operational message
   Ax18_DB2_524 : BOOL  := TRUE;	// error message
   Ax18_DB2_525 : BOOL ;	// operational message
   Ax19_DB2_526 : BOOL  := TRUE;	// error message
   Ax19_DB2_527 : BOOL ;	// operational message
   Ax20_DB2_528 : BOOL  := TRUE;	// error message
   Ax20_DB2_529 : BOOL ;	// operational message
   Ax21_DB2_530 : BOOL  := TRUE;	// error message
   Ax21_DB2_531 : BOOL ;	// operational message
   Ax22_DB2_532 : BOOL  := TRUE;	// error message
   Ax22_DB2_533 : BOOL ;	// operational message
   Ax23_DB2_534 : BOOL  := TRUE;	// error message
   Ax23_DB2_535 : BOOL ;	// operational message
   Ax24_DB2_536 : BOOL  := TRUE;	// error message
   Ax24_DB2_537 : BOOL ;	// operational message
   Ax25_DB2_538 : BOOL  := TRUE;	// error message
   Ax25_DB2_539 : BOOL ;	// operational message
   Ax26_DB2_540 : BOOL  := TRUE;	// error message
   Ax26_DB2_541 : BOOL ;	// operational message
   Ax27_DB2_542 : BOOL  := TRUE;	// error message
   Ax27_DB2_543 : BOOL ;	// operational message
   Ax28_DB2_544 : BOOL  := TRUE;	// error message
   Ax28_DB2_545 : BOOL ;	// operational message
   Ax29_DB2_546 : BOOL  := TRUE;	// error message
   Ax29_DB2_547 : BOOL ;	// operational message
   Ax30_DB2_548 : BOOL  := TRUE;	// error message
   Ax30_DB2_549 : BOOL ;	// operational message
   Ax31_DB2_550 : BOOL  := TRUE;	// error message
   Ax31_DB2_551 : BOOL ;	// operational message
   Ax32_DB2_552 : BOOL  := TRUE;	// error message
   Ax32_DB2_553 : BOOL ;	// operational message
   User0_DB2_554 : BOOL  := TRUE;	// (32 User data area ever 8 Bit):  error message
   User0_DB2_555 : BOOL  := TRUE;	// UserDataArea 0, DB2.DBB555; error message
   User0_DB2_556 : BOOL  := TRUE;	// error message
   User0_DB2_557 : BOOL  := TRUE;	// error message
   User0_DB2_558 : BOOL ;	// operational message
   User0_DB2_559 : BOOL ;	// operational message
   User0_DB2_560 : BOOL ;	// operational message
   User0_DB2_561 : BOOL ;	// operational message
   User1_DB2_562 : BOOL  := TRUE;	// UserDataArea 1, DB2.DBB562; error message
   User1_DB2_563 : BOOL  := TRUE;	// error message
   User1_DB2_564 : BOOL  := TRUE;	// error message
   User1_DB2_565 : BOOL  := TRUE;	// error message
   User1_DB2_566 : BOOL ;	// operational message
   User1_DB2_567 : BOOL ;	// operational message
   User1_DB2_568 : BOOL ;	// operational message
   User1_DB2_569 : BOOL ;	// operational message
   User2_DB2_570 : BOOL  := TRUE;	// UserDataArea 2, DB2.DBB570; error message
   User2_DB2_571 : BOOL  := TRUE;	// error message
   User2_DB2_572 : BOOL  := TRUE;	// error message
   User2_DB2_573 : BOOL  := TRUE;	// error message
   User2_DB2_574 : BOOL ;	// operational message
   User2_DB2_575 : BOOL ;	// operational message
   User2_DB2_576 : BOOL ;	// operational message
   User2_DB2_577 : BOOL ;	// operational message
   User3_DB2_578 : BOOL  := TRUE;	// UserDataArea 3, DB2.DBB578; error message
   User3_DB2_579 : BOOL  := TRUE;	// error message
   User3_DB2_580 : BOOL  := TRUE;	// error message
   User3_DB2_581 : BOOL  := TRUE;	// error message
   User3_DB2_582 : BOOL ;	// operational message
   User3_DB2_583 : BOOL ;	// operational message
   User3_DB2_584 : BOOL ;	// operational message
   User3_DB2_585 : BOOL ;	// operational message
   User4_DB2_586 : BOOL  := TRUE;	// UserDataArea 4, DB2.DBB586; error message
   User4_DB2_587 : BOOL  := TRUE;	// error message
   User4_DB2_588 : BOOL  := TRUE;	// error message
   User4_DB2_589 : BOOL  := TRUE;	// error message
   User4_DB2_590 : BOOL ;	// operational message
   User4_DB2_591 : BOOL ;	// operational message
   User4_DB2_592 : BOOL ;	// operational message
   User4_DB2_593 : BOOL ;	// operational message
   User5_DB2_594 : BOOL  := TRUE;	// UserDataArea 5, DB2.DBB594; error message
   User5_DB2_595 : BOOL  := TRUE;	// error message
   User5_DB2_596 : BOOL  := TRUE;	// error message
   User5_DB2_597 : BOOL  := TRUE;	// error message
   User5_DB2_598 : BOOL ;	// operational message
   User5_DB2_599 : BOOL ;	// operational message
   User5_DB2_600 : BOOL ;	// operational message
   User5_DB2_601 : BOOL ;	// operational message
   User6_DB2_602 : BOOL  := TRUE;	// UserDataArea 6, DB2.DBB602; error message
   User6_DB2_603 : BOOL  := TRUE;	// error message
   User6_DB2_604 : BOOL  := TRUE;	// error message
   User6_DB2_605 : BOOL  := TRUE;	// error message
   User6_DB2_606 : BOOL ;	// operational message
   User6_DB2_607 : BOOL ;	// operational message
   User6_DB2_608 : BOOL ;	// operational message
   User6_DB2_609 : BOOL ;	// operational message
   User7_DB2_610 : BOOL  := TRUE;	// UserDataArea 7, DB2.DBB610; error message
   User7_DB2_611 : BOOL  := TRUE;	// error message
   User7_DB2_612 : BOOL  := TRUE;	// error message
   User7_DB2_613 : BOOL  := TRUE;	// error message
   User7_DB2_614 : BOOL ;	// operational message
   User7_DB2_615 : BOOL ;	// operational message
   User7_DB2_616 : BOOL ;	// operational message
   User7_DB2_617 : BOOL ;	// operational message
   User8_DB2_618 : BOOL  := TRUE;	// UserDataArea 8, DB2.DBB618; error message
   User8_DB2_619 : BOOL  := TRUE;	// error message
   User8_DB2_620 : BOOL  := TRUE;	// error message
   User8_DB2_621 : BOOL  := TRUE;	// error message
   User8_DB2_622 : BOOL ;	// operational message
   User8_DB2_623 : BOOL ;	// operational message
   User8_DB2_624 : BOOL ;	// operational message
   User8_DB2_625 : BOOL ;	// operational message
   User9_DB2_626 : BOOL  := TRUE;	// UserDataArea 9, DB2.DBB626; error message
   User9_DB2_627 : BOOL  := TRUE;	// error message
   User9_DB2_628 : BOOL  := TRUE;	// error message
   User9_DB2_629 : BOOL  := TRUE;	// error message
   User9_DB2_630 : BOOL ;	// operational message
   User9_DB2_631 : BOOL ;	// operational message
   User9_DB2_632 : BOOL ;	// operational message
   User9_DB2_633 : BOOL ;	// operational message
   User10_DB2_634 : BOOL  := TRUE;	// UserDataArea 10, DB2.DBB634; error message
   User10_DB2_635 : BOOL  := TRUE;	// error message
   User10_DB2_636 : BOOL  := TRUE;	// error message
   User10_DB2_637 : BOOL  := TRUE;	// error message
   User10_DB2_638 : BOOL ;	// operational message
   User10_DB2_639 : BOOL ;	// operational message
   User10_DB2_640 : BOOL ;	// operational message
   User10_DB2_641 : BOOL ;	// operational message
   User11_DB2_642 : BOOL  := TRUE;	// UserDataArea 11, DB2.DBB642; error message
   User11_DB2_643 : BOOL  := TRUE;	// error message
   User11_DB2_644 : BOOL  := TRUE;	// error message
   User11_DB2_645 : BOOL  := TRUE;	// error message
   User11_DB2_646 : BOOL ;	// operational message
   User11_DB2_647 : BOOL ;	// operational message
   User11_DB2_648 : BOOL ;	// operational message
   User11_DB2_649 : BOOL ;	// operational message
   User12_DB2_650 : BOOL  := TRUE;	// UserDataArea 12, DB2.DBB650; error message
   User12_DB2_651 : BOOL  := TRUE;	// error message
   User12_DB2_652 : BOOL  := TRUE;	// error message
   User12_DB2_653 : BOOL  := TRUE;	// error message
   User12_DB2_654 : BOOL ;	// operational message
   User12_DB2_655 : BOOL ;	// operational message
   User12_DB2_656 : BOOL ;	// operational message
   User12_DB2_657 : BOOL ;	// operational message
   User13_DB2_658 : BOOL  := TRUE;	// UserDataArea 13, DB2.DBB658; error message
   User13_DB2_659 : BOOL  := TRUE;	// error message
   User13_DB2_660 : BOOL  := TRUE;	// error message
   User13_DB2_661 : BOOL  := TRUE;	// error message
   User13_DB2_662 : BOOL ;	// operational message
   User13_DB2_663 : BOOL ;	// operational message
   User13_DB2_664 : BOOL ;	// operational message
   User13_DB2_665 : BOOL ;	// operational message
   User14_DB2_666 : BOOL  := TRUE;	// UserDataArea 14, DB2.DBB666; error message
   User14_DB2_667 : BOOL  := TRUE;	// error message
   User14_DB2_668 : BOOL  := TRUE;	// error message
   User14_DB2_669 : BOOL  := TRUE;	// error message
   User14_DB2_670 : BOOL ;	// operational message
   User14_DB2_671 : BOOL ;	// operational message
   User14_DB2_672 : BOOL ;	// operational message
   User14_DB2_673 : BOOL ;	// operational message
   User15_DB2_674 : BOOL  := TRUE;	// UserDataArea 15, DB2.DBB674; error message
   User15_DB2_675 : BOOL  := TRUE;	// error message
   User15_DB2_676 : BOOL  := TRUE;	// error message
   User15_DB2_677 : BOOL  := TRUE;	// error message
   User15_DB2_678 : BOOL ;	// operational message
   User15_DB2_679 : BOOL ;	// operational message
   User15_DB2_680 : BOOL ;	// operational message
   User15_DB2_681 : BOOL ;	// operational message
   User16_DB2_682 : BOOL  := TRUE;	// UserDataArea 16, DB2.DBB682; error message
   User16_DB2_683 : BOOL  := TRUE;	// error message
   User16_DB2_684 : BOOL  := TRUE;	// error message
   User16_DB2_685 : BOOL  := TRUE;	// error message
   User16_DB2_686 : BOOL ;	// operational message
   User16_DB2_687 : BOOL ;	// operational message
   User16_DB2_688 : BOOL ;	// operational message
   User16_DB2_689 : BOOL ;	// operational message
   User17_DB2_690 : BOOL  := TRUE;	// UserDataArea 17, DB2.DBB690; error message
   User17_DB2_691 : BOOL  := TRUE;	// error message
   User17_DB2_692 : BOOL  := TRUE;	// error message
   User17_DB2_693 : BOOL  := TRUE;	// error message
   User17_DB2_694 : BOOL ;	// operational message
   User17_DB2_695 : BOOL ;	// operational message
   User17_DB2_696 : BOOL ;	// operational message
   User17_DB2_697 : BOOL ;	// operational message
   User18_DB2_698 : BOOL  := TRUE;	// UserDataArea 18, DB2.DBB698; error message
   User18_DB2_699 : BOOL  := TRUE;	// error message
   User18_DB2_700 : BOOL  := TRUE;	// error message
   User18_DB2_701 : BOOL  := TRUE;	// error message
   User18_DB2_702 : BOOL ;	// operational message
   User18_DB2_703 : BOOL ;	// operational message
   User18_DB2_704 : BOOL ;	// operational message
   User18_DB2_705 : BOOL ;	// operational message
   User19_DB2_706 : BOOL  := TRUE;	// UserDataArea 19, DB2.DBB706; error message
   User19_DB2_707 : BOOL  := TRUE;	// error message
   User19_DB2_708 : BOOL  := TRUE;	// error message
   User19_DB2_709 : BOOL  := TRUE;	// error message
   User19_DB2_710 : BOOL ;	// operational message
   User19_DB2_711 : BOOL ;	// operational message
   User19_DB2_712 : BOOL ;	// operational message
   User19_DB2_713 : BOOL ;	// operational message
   User20_DB2_714 : BOOL  := TRUE;	// UserDataArea 20, DB2.DBB714; error message
   User20_DB2_715 : BOOL  := TRUE;	// error message
   User20_DB2_716 : BOOL  := TRUE;	// error message
   User20_DB2_717 : BOOL  := TRUE;	// error message
   User20_DB2_718 : BOOL ;	// operational message
   User20_DB2_719 : BOOL ;	// operational message
   User20_DB2_720 : BOOL ;	// operational message
   User20_DB2_721 : BOOL ;	// operational message
   User21_DB2_722 : BOOL  := TRUE;	// UserDataArea 21, DB2.DBB722; error message
   User21_DB2_723 : BOOL  := TRUE;	// error message
   User21_DB2_724 : BOOL  := TRUE;	// error message
   User21_DB2_725 : BOOL  := TRUE;	// error message
   User21_DB2_726 : BOOL ;	// operational message
   User21_DB2_727 : BOOL ;	// operational message
   User21_DB2_728 : BOOL ;	// operational message
   User21_DB2_729 : BOOL ;	// operational message
   User22_DB2_730 : BOOL  := TRUE;	// UserDataArea 22, DB2.DBB730; error message
   User22_DB2_731 : BOOL  := TRUE;	// error message
   User22_DB2_732 : BOOL  := TRUE;	// error message
   User22_DB2_733 : BOOL  := TRUE;	// error message
   User22_DB2_734 : BOOL ;	// operational message
   User22_DB2_735 : BOOL ;	// operational message
   User22_DB2_736 : BOOL ;	// operational message
   User22_DB2_737 : BOOL ;	// operational message
   User23_DB2_738 : BOOL  := TRUE;	// UserDataArea 23, DB2.DBB738; error message
   User23_DB2_739 : BOOL  := TRUE;	// error message
   User23_DB2_740 : BOOL  := TRUE;	// error message
   User23_DB2_741 : BOOL  := TRUE;	// error message
   User23_DB2_742 : BOOL ;	// operational message
   User23_DB2_743 : BOOL ;	// operational message
   User23_DB2_744 : BOOL ;	// operational message
   User23_DB2_745 : BOOL ;	// operational message
   User24_DB2_746 : BOOL  := TRUE;	// UserDataArea 24, DB2.DBB746; error message
   User24_DB2_747 : BOOL  := TRUE;	// error message
   User24_DB2_748 : BOOL  := TRUE;	// error message
   User24_DB2_749 : BOOL  := TRUE;	// error message
   User24_DB2_750 : BOOL ;	// operational message
   User24_DB2_751 : BOOL ;	// operational message
   User24_DB2_752 : BOOL ;	// operational message
   User24_DB2_753 : BOOL ;	// operational message
   User25_DB2_754 : BOOL  := TRUE;	// UserDataArea 25, DB2.DBB754; error message
   User25_DB2_755 : BOOL  := TRUE;	// error message
   User25_DB2_756 : BOOL  := TRUE;	// error message
   User25_DB2_757 : BOOL  := TRUE;	// error message
   User25_DB2_758 : BOOL ;	// operational message
   User25_DB2_759 : BOOL ;	// operational message
   User25_DB2_760 : BOOL ;	// operational message
   User25_DB2_761 : BOOL ;	// operational message
   User26_DB2_762 : BOOL  := TRUE;	// UserDataArea 26, DB2.DBB762; error message
   User26_DB2_763 : BOOL  := TRUE;	// error message
   User26_DB2_764 : BOOL  := TRUE;	// error message
   User26_DB2_765 : BOOL  := TRUE;	// error message
   User26_DB2_766 : BOOL ;	// operational message
   User26_DB2_767 : BOOL ;	// operational message
   User26_DB2_768 : BOOL ;	// operational message
   User26_DB2_769 : BOOL ;	// operational message
   User27_DB2_770 : BOOL  := TRUE;	// UserDataArea 27, DB2.DBB770; error message
   User27_DB2_771 : BOOL  := TRUE;	// error message
   User27_DB2_772 : BOOL  := TRUE;	// error message
   User27_DB2_773 : BOOL  := TRUE;	// error message
   User27_DB2_774 : BOOL ;	// operational message
   User27_DB2_775 : BOOL ;	// operational message
   User27_DB2_776 : BOOL ;	// operational message
   User27_DB2_777 : BOOL ;	// operational message
   User28_DB2_778 : BOOL  := TRUE;	// UserDataArea 28, DB2.DBB778; error message
   User28_DB2_779 : BOOL  := TRUE;	// error message
   User28_DB2_780 : BOOL  := TRUE;	// error message
   User28_DB2_781 : BOOL  := TRUE;	// error message
   User28_DB2_782 : BOOL ;	// operational message
   User28_DB2_783 : BOOL ;	// operational message
   User28_DB2_784 : BOOL ;	// operational message
   User28_DB2_785 : BOOL ;	// operational message
   User29_DB2_786 : BOOL  := TRUE;	// UserDataArea 29, DB2.DBB786; error message
   User29_DB2_787 : BOOL  := TRUE;	// error message
   User29_DB2_788 : BOOL  := TRUE;	// error message
   User29_DB2_789 : BOOL  := TRUE;	// error message
   User29_DB2_790 : BOOL ;	// operational message
   User29_DB2_791 : BOOL ;	// operational message
   User29_DB2_792 : BOOL ;	// operational message
   User29_DB2_793 : BOOL ;	// operational message
   User30_DB2_794 : BOOL  := TRUE;	// UserDataArea 30, DB2.DBB794; error message
   User30_DB2_795 : BOOL  := TRUE;	// error message
   User30_DB2_796 : BOOL  := TRUE;	// error message
   User30_DB2_797 : BOOL  := TRUE;	// error message
   User30_DB2_798 : BOOL ;	// operational message
   User30_DB2_799 : BOOL ;	// operational message
   User30_DB2_800 : BOOL ;	// operational message
   User30_DB2_801 : BOOL ;	// operational message
   User31_DB2_802 : BOOL  := TRUE;	// UserDataArea 31, DB2.DBB802; error message
   User31_DB2_803 : BOOL  := TRUE;	// error message
   User31_DB2_804 : BOOL  := TRUE;	// error message
   User31_DB2_805 : BOOL  := TRUE;	// error message
   User31_DB2_806 : BOOL ;	// operational message
   User31_DB2_807 : BOOL ;	// operational message
   User31_DB2_808 : BOOL ;	// operational message
   User31_DB2_809 : BOOL ;	// operational message
   Bit62_4 : BOOL ;	// reserved
   Bit62_5 : BOOL ;	// reserved
   Bit62_6 : BOOL ;	// reserved
   Bit62_7 : BOOL ;	// reserved
   Byte63 : BYTE ;	// reserved
   Word64 : WORD ;	// reserved
   Word66 : WORD ;	// reserved
   Word68 : WORD ;	// reserved
   Word70 : WORD ;	// reserved
   UserDek2No : ARRAY  [0 .. 31 ] OF // UserDek2No: Value 0..9 possible
   BYTE  := B#16#0;
  END_STRUCT ;	
BEGIN
   Ch1_DB2_310 := TRUE;
   Ch1_DB2_312 := TRUE;
   Ch1_DB2_313 := TRUE;
   Ch1_DB2_316 := TRUE;
   Ch1_DB2_317 := TRUE;
   Ch1_DB2_320 := TRUE;
   Ch1_DB2_322 := TRUE;
   Ch1_DB2_324 := TRUE;
   Ch1_DB2_326 := TRUE;
   Ch2_DB2_328 := TRUE;
   Ch2_DB2_330 := TRUE;
   Ch2_DB2_331 := TRUE;
   Ch2_DB2_334 := TRUE;
   Ch2_DB2_335 := TRUE;
   Ch2_DB2_338 := TRUE;
   Ch2_DB2_340 := TRUE;
   Ch2_DB2_342 := TRUE;
   Ch2_DB2_344 := TRUE;
   Ch3_DB2_346 := TRUE;
   Ch3_DB2_348 := TRUE;
   Ch3_DB2_349 := TRUE;
   Ch3_DB2_352 := TRUE;
   Ch3_DB2_353 := TRUE;
   Ch3_DB2_356 := TRUE;
   Ch3_DB2_358 := TRUE;
   Ch3_DB2_360 := TRUE;
   Ch3_DB2_362 := TRUE;
   Ch4_DB2_364 := TRUE;
   Ch4_DB2_366 := TRUE;
   Ch4_DB2_367 := TRUE;
   Ch4_DB2_370 := TRUE;
   Ch4_DB2_371 := TRUE;
   Ch4_DB2_374 := TRUE;
   Ch4_DB2_376 := TRUE;
   Ch4_DB2_378 := TRUE;
   Ch4_DB2_380 := TRUE;
   Ch5_DB2_382 := TRUE;
   Ch5_DB2_384 := TRUE;
   Ch5_DB2_385 := TRUE;
   Ch5_DB2_388 := TRUE;
   Ch5_DB2_389 := TRUE;
   Ch5_DB2_392 := TRUE;
   Ch5_DB2_394 := TRUE;
   Ch5_DB2_396 := TRUE;
   Ch5_DB2_398 := TRUE;
   Ch6_DB2_400 := TRUE;
   Ch6_DB2_402 := TRUE;
   Ch6_DB2_403 := TRUE;
   Ch6_DB2_406 := TRUE;
   Ch6_DB2_407 := TRUE;
   Ch6_DB2_410 := TRUE;
   Ch6_DB2_412 := TRUE;
   Ch6_DB2_414 := TRUE;
   Ch6_DB2_416 := TRUE;
   Ch7_DB2_418 := TRUE;
   Ch7_DB2_420 := TRUE;
   Ch7_DB2_421 := TRUE;
   Ch7_DB2_424 := TRUE;
   Ch7_DB2_425 := TRUE;
   Ch7_DB2_428 := TRUE;
   Ch7_DB2_430 := TRUE;
   Ch7_DB2_432 := TRUE;
   Ch7_DB2_434 := TRUE;
   Ch8_DB2_436 := TRUE;
   Ch8_DB2_438 := TRUE;
   Ch8_DB2_439 := TRUE;
   Ch8_DB2_442 := TRUE;
   Ch8_DB2_443 := TRUE;
   Ch8_DB2_446 := TRUE;
   Ch8_DB2_448 := TRUE;
   Ch8_DB2_450 := TRUE;
   Ch8_DB2_452 := TRUE;
   Ch9_DB2_454 := TRUE;
   Ch9_DB2_456 := TRUE;
   Ch9_DB2_457 := TRUE;
   Ch9_DB2_460 := TRUE;
   Ch9_DB2_461 := TRUE;
   Ch9_DB2_464 := TRUE;
   Ch9_DB2_466 := TRUE;
   Ch9_DB2_468 := TRUE;
   Ch9_DB2_470 := TRUE;
   Ch10_DB2_472 := TRUE;
   Ch10_DB2_474 := TRUE;
   Ch10_DB2_475 := TRUE;
   Ch10_DB2_478 := TRUE;
   Ch10_DB2_479 := TRUE;
   Ch10_DB2_482 := TRUE;
   Ch10_DB2_484 := TRUE;
   Ch10_DB2_486 := TRUE;
   Ch10_DB2_488 := TRUE;
   Ax1_DB2_490 := TRUE;
   Ax2_DB2_492 := TRUE;
   Ax3_DB2_494 := TRUE;
   Ax4_DB2_496 := TRUE;
   Ax5_DB2_498 := TRUE;
   Ax6_DB2_500 := TRUE;
   Ax7_DB2_502 := TRUE;
   Ax8_DB2_504 := TRUE;
   Ax9_DB2_506 := TRUE;
   Ax10_DB2_508 := TRUE;
   Ax11_DB2_510 := TRUE;
   Ax12_DB2_512 := TRUE;
   Ax13_DB2_514 := TRUE;
   Ax14_DB2_516 := TRUE;
   Ax15_DB2_518 := TRUE;
   Ax16_DB2_520 := TRUE;
   Ax17_DB2_522 := TRUE;
   Ax18_DB2_524 := TRUE;
   Ax19_DB2_526 := TRUE;
   Ax20_DB2_528 := TRUE;
   Ax21_DB2_530 := TRUE;
   Ax22_DB2_532 := TRUE;
   Ax23_DB2_534 := TRUE;
   Ax24_DB2_536 := TRUE;
   Ax25_DB2_538 := TRUE;
   Ax26_DB2_540 := TRUE;
   Ax27_DB2_542 := TRUE;
   Ax28_DB2_544 := TRUE;
   Ax29_DB2_546 := TRUE;
   Ax30_DB2_548 := TRUE;
   Ax31_DB2_550 := TRUE;
   Ax32_DB2_552 := TRUE;
   User0_DB2_554 := TRUE;
   User0_DB2_555 := TRUE;
   User0_DB2_556 := TRUE;
   User0_DB2_557 := TRUE;
   User1_DB2_562 := TRUE;
   User1_DB2_563 := TRUE;
   User1_DB2_564 := TRUE;
   User1_DB2_565 := TRUE;
   User2_DB2_570 := TRUE;
   User2_DB2_571 := TRUE;
   User2_DB2_572 := TRUE;
   User2_DB2_573 := TRUE;
   User3_DB2_578 := TRUE;
   User3_DB2_579 := TRUE;
   User3_DB2_580 := TRUE;
   User3_DB2_581 := TRUE;
   User4_DB2_586 := TRUE;
   User4_DB2_587 := TRUE;
   User4_DB2_588 := TRUE;
   User4_DB2_589 := TRUE;
   User5_DB2_594 := TRUE;
   User5_DB2_595 := TRUE;
   User5_DB2_596 := TRUE;
   User5_DB2_597 := TRUE;
   User6_DB2_602 := TRUE;
   User6_DB2_603 := TRUE;
   User6_DB2_604 := TRUE;
   User6_DB2_605 := TRUE;
   User7_DB2_610 := TRUE;
   User7_DB2_611 := TRUE;
   User7_DB2_612 := TRUE;
   User7_DB2_613 := TRUE;
   User8_DB2_618 := TRUE;
   User8_DB2_619 := TRUE;
   User8_DB2_620 := TRUE;
   User8_DB2_621 := TRUE;
   User9_DB2_626 := TRUE;
   User9_DB2_627 := TRUE;
   User9_DB2_628 := TRUE;
   User9_DB2_629 := TRUE;
   User10_DB2_634 := TRUE;
   User10_DB2_635 := TRUE;
   User10_DB2_636 := TRUE;
   User10_DB2_637 := TRUE;
   User11_DB2_642 := TRUE;
   User11_DB2_643 := TRUE;
   User11_DB2_644 := TRUE;
   User11_DB2_645 := TRUE;
   User12_DB2_650 := TRUE;
   User12_DB2_651 := TRUE;
   User12_DB2_652 := TRUE;
   User12_DB2_653 := TRUE;
   User13_DB2_658 := TRUE;
   User13_DB2_659 := TRUE;
   User13_DB2_660 := TRUE;
   User13_DB2_661 := TRUE;
   User14_DB2_666 := TRUE;
   User14_DB2_667 := TRUE;
   User14_DB2_668 := TRUE;
   User14_DB2_669 := TRUE;
   User15_DB2_674 := TRUE;
   User15_DB2_675 := TRUE;
   User15_DB2_676 := TRUE;
   User15_DB2_677 := TRUE;
   User16_DB2_682 := TRUE;
   User16_DB2_683 := TRUE;
   User16_DB2_684 := TRUE;
   User16_DB2_685 := TRUE;
   User17_DB2_690 := TRUE;
   User17_DB2_691 := TRUE;
   User17_DB2_692 := TRUE;
   User17_DB2_693 := TRUE;
   User18_DB2_698 := TRUE;
   User18_DB2_699 := TRUE;
   User18_DB2_700 := TRUE;
   User18_DB2_701 := TRUE;
   User19_DB2_706 := TRUE;
   User19_DB2_707 := TRUE;
   User19_DB2_708 := TRUE;
   User19_DB2_709 := TRUE;
   User20_DB2_714 := TRUE;
   User20_DB2_715 := TRUE;
   User20_DB2_716 := TRUE;
   User20_DB2_717 := TRUE;
   User21_DB2_722 := TRUE;
   User21_DB2_723 := TRUE;
   User21_DB2_724 := TRUE;
   User21_DB2_725 := TRUE;
   User22_DB2_730 := TRUE;
   User22_DB2_731 := TRUE;
   User22_DB2_732 := TRUE;
   User22_DB2_733 := TRUE;
   User23_DB2_738 := TRUE;
   User23_DB2_739 := TRUE;
   User23_DB2_740 := TRUE;
   User23_DB2_741 := TRUE;
   User24_DB2_746 := TRUE;
   User24_DB2_747 := TRUE;
   User24_DB2_748 := TRUE;
   User24_DB2_749 := TRUE;
   User25_DB2_754 := TRUE;
   User25_DB2_755 := TRUE;
   User25_DB2_756 := TRUE;
   User25_DB2_757 := TRUE;
   User26_DB2_762 := TRUE;
   User26_DB2_763 := TRUE;
   User26_DB2_764 := TRUE;
   User26_DB2_765 := TRUE;
   User27_DB2_770 := TRUE;
   User27_DB2_771 := TRUE;
   User27_DB2_772 := TRUE;
   User27_DB2_773 := TRUE;
   User28_DB2_778 := TRUE;
   User28_DB2_779 := TRUE;
   User28_DB2_780 := TRUE;
   User28_DB2_781 := TRUE;
   User29_DB2_786 := TRUE;
   User29_DB2_787 := TRUE;
   User29_DB2_788 := TRUE;
   User29_DB2_789 := TRUE;
   User30_DB2_794 := TRUE;
   User30_DB2_795 := TRUE;
   User30_DB2_796 := TRUE;
   User30_DB2_797 := TRUE;
   User31_DB2_802 := TRUE;
   User31_DB2_803 := TRUE;
   User31_DB2_804 := TRUE;
   User31_DB2_805 := TRUE;
END_DATA_BLOCK

DATA_BLOCK "gp_par"	// DB 7
TITLE = Parameters for Baseprogram
AUTHOR : NUMERIK
FAMILY : _800D
NAME : Basics
VERSION : 4.5
"RUN_UP"
BEGIN
END_DATA_BLOCK

DATA_BLOCK DB 8
AUTHOR : NUMERIK
FAMILY : _800D
NAME : Basics
VERSION : 4.5
  STRUCT
   Fc19_1 : ARRAY  [0 .. 3 ] OF BYTE ;
   Res0 : ARRAY  [0 .. 3 ] OF BYTE ;
   plData : ARRAY  [8 .. 43 ] OF BYTE ;
   TestAuto : BYTE ;
   FirstCycle : BYTE ;
   Res4 : WORD ;
   Res5 : BYTE ;
   IsFb15Correct : BYTE ;
   Res6 : ARRAY  [50 .. 61 ] OF BYTE ;
   Fc19_2 : ARRAY  [0 .. 3 ] OF BYTE ;
   Res8 : ARRAY  [66 .. 81 ] OF BYTE ;
   S7_error_id : WORD ;
   S7_error_param : WORD ;
   S7_error_adr : DWORD ;
   MinCycleTime : INT ;
   AdaptTime : INT ;
   ActCycleTime : INT ;
  END_STRUCT ;	
BEGIN
END_DATA_BLOCK

DATA_BLOCK DB 15
AUTHOR : NUMERIK
FAMILY : _800D
NAME : Bas_Com
VERSION : 4.5
  STRUCT
   fifoFull : BOOL ;
   readOffset : BYTE ;
   writeOffset : BYTE ;
   filler : BYTE ;
   Fifo : ARRAY  [1 .. 10 ] OF BYTE ;
   pduRefArr : ARRAY  [1 .. 12 ] OF //Little Endian Werte
   STRUCT
    diNo : WORD ;
    diPartLen : WORD ;
    PdiBeg : DWORD ;
   END_STRUCT ;
  END_STRUCT ;	
BEGIN
END_DATA_BLOCK

// DB 16: know-how protected block, not included

DATA_BLOCK "SPL"	// DB 18
TITLE = SPL dataarea
AUTHOR : NUMERIK
FAMILY : _800D
NAME : Basics
VERSION : 4.5
  STRUCT
   INSEP_VALID : ARRAY  [1 .. 8 ] OF BOOL ;	//used external SPL-Inputbytes(HW)
   OUTSEP_VALID : ARRAY  [1 .. 8 ] OF BOOL ;	//used external SPL-Outputbytes(HW)
   INSEP_ADDR : ARRAY  [1 .. 8 ] OF INT ;	//Addresses external SPL-Inputbytes(HW)
   OUTSEP_ADDR : ARRAY  [1 .. 8 ] OF INT ;	//Addresses external SPL-Outputbytes(HW)
   SPL_READY : BOOL ;	//setup finished
   STOP_MODE : BOOL ;	//0= Stop D, 1=Stop E
   SPL_DATA : STRUCT
    INSEP : ARRAY  [1 .. 64 ] OF BOOL ;
    OUTSEP : ARRAY  [1 .. 64 ] OF BOOL ;
    INSIP : ARRAY  [1 .. 64 ] OF BOOL ;
    OUTSIP : ARRAY  [1 .. 64 ] OF BOOL ;
    MARKERSIP : ARRAY  [1 .. 64 ] OF BOOL ;
   END_STRUCT ;
   SPL_DELTA : STRUCT 	//edge difference NCK - PLC for Diagnostic
    INSEP : ARRAY  [1 .. 64 ] OF BOOL ;
    OUTSEP : ARRAY  [1 .. 64 ] OF BOOL ;
    INSIP : ARRAY  [1 .. 64 ] OF BOOL ;
    OUTSIP : ARRAY  [1 .. 64 ] OF BOOL ;
    MARKERSIP : ARRAY  [1 .. 64 ] OF BOOL ;
   END_STRUCT ;
   CMDSI : BOOL ;	//multiplication of Timeout Value by Factor 10
   CMDSI_R1 : BOOL ;	//for future use
   CMDSI_R2 : BOOL ;	//for future use
   CMDSI_R3 : BOOL ;	//for future use
   CMDSI_R4 : BOOL ;	//for future use
   CMDSI_R5 : BOOL ;	//for future use
   CMDSI_R6 : BOOL ;	//for future use
   CMDSI_R7 : BOOL ;	//for future use
   STATUS_R0 : BOOL ;	//for future use
   STATUS_R1 : BOOL ;	//for future use
   PS_COMM_ERR : BOOL ;	//PROFIsafe Communication Error
   STATUS_R3 : BOOL ;	//for future use
   IBN_FAULT : BOOL ;	//CDC error: SPL protection status
   COMM_TO : BOOL ;	//Communication Timeout
   STOP_FROM_NC : BOOL ;	//NCK signals a stop to the PLC.
   STATUS_R7 : BOOL ;	//for future use
   STATSI : DINT ;	//Status: 0 - no error, 1 - 320 error number
   LEVELSI : DINT ;	//stacklevel SPL-KDV for Diagnostic
   PLCSIOUT : ARRAY  [1 .. 32 ] OF BOOL ;	//Single Channel Signals from NCK
   PLCSIIN : ARRAY  [1 .. 32 ] OF BOOL ;	//Single Channel Signals to NCK
   SPL_STATUS : ARRAY  [1 .. 16 ] OF BOOL ;	//SPL Status from NCK
   INSEP_PROFISAFE : ARRAY  [1 .. 8 ] OF BOOL ;	//external SPL-Inputbytes(HW) with PROFIsafe Slaves
   OUTSEP_PROFISAFE : ARRAY  [1 .. 8 ] OF BOOL ;	//external SPL-Outputbytes(HW) with PROFIsafe Slaves
   NoOfAxisPerBlock : ARRAY  [1 .. 8 ] OF BYTE ;	//Pointer and Tables for Teststop
   BlockPointer : ARRAY  [1 .. 8 ] OF BYTE ;
   AxisTable : ARRAY  [1 .. 31 ] OF BYTE ;
   FSDP : ARRAY  [1 .. 3 ] OF STRUCT
    ERR_REAC : INT ;	// IN: Error reaction
    ERROR : BOOL ;	// OUT: 1=Communication error
    SUBS_ON : BOOL ;	// OUT: 1=Receiver outputs fail-safe values
    DIAG : WORD ;	// OUT: Service information
    RETVAL14 : WORD ;	// OUT: Error code of SFC 14
    RETVAL15 : WORD ;	// OUT: Error code of SFC 15
   END_STRUCT ;
   FRDP : ARRAY  [1 .. 3 ] OF STRUCT
    SUBS : ARRAY  [0 .. 15 ] OF BOOL ;	// IN: Fail-safe value for receive data BOOL 00 ... BOOL 15
    ERR_REAC : INT ;	// IN: Error reaction
    ACK_REI : BOOL ;	// IN: 1=Acknowledgment for reintegration of send data following communication er
    RES1 : BOOL ;	//Reserved
    RES2 : BOOL ;	//Reserved
    RES3 : BOOL ;	//Reserved
    RES4 : BOOL ;	//Reserved
    RES5 : BOOL ;	//Reserved
    RES6 : BOOL ;	//Reserved
    RES7 : BOOL ;	//Reserved
    ERROR : BOOL ;	// OUT: 1=Communication error
    SUBS_ON : BOOL ;	// OUT: 1=Fail-safe values are output
    ACK_REQ : BOOL ;	// OUT: 1=Acknowledgment for reintegration of send data required
    SENDMODE : BOOL ;	// OUT: 1=F_CPU with F_SENDDP in deactivated safety mode
    DIAG : WORD ;	// OUT: Service information
    RETVAL14 : WORD ;	// OUT: Error code of SFC 14
    RETVAL15 : WORD ;	// OUT: Error code of SFC 15
   END_STRUCT ;
   SPL_USER_DATA : ARRAY  [0 .. 3 ] OF DWORD ;
   SPL_DATA_HF : STRUCT
    INSEP : ARRAY  [65 .. 192 ] OF BOOL ;
    OUTSEP : ARRAY  [65 .. 192 ] OF BOOL ;
    INSIP : ARRAY  [65 .. 192 ] OF BOOL ;
    OUTSIP : ARRAY  [65 .. 192 ] OF BOOL ;
    MARKERSIP : ARRAY  [65 .. 192 ] OF BOOL ;
   END_STRUCT ;
   SPL_DELTA_HF : STRUCT 	//edge difference NCK - PLC for Diagnostic
    INSEP : ARRAY  [65 .. 192 ] OF BOOL ;
    OUTSEP : ARRAY  [65 .. 192 ] OF BOOL ;
    INSIP : ARRAY  [65 .. 192 ] OF BOOL ;
    OUTSIP : ARRAY  [65 .. 192 ] OF BOOL ;
    MARKERSIP : ARRAY  [65 .. 192 ] OF BOOL ;
   END_STRUCT ;
   PLCSIOUT_HF : ARRAY  [33 .. 96 ] OF BOOL ;	//Single Channel Signals from NCK
   PLCSIIN_HF : ARRAY  [33 .. 96 ] OF BOOL ;	//Single Channel Signals to NCK
  END_STRUCT ;	
BEGIN
END_DATA_BLOCK

DATA_BLOCK "MMC"	// DB 19
VERSION : 0.0
BEGIN
// 404 bytes; values not shown
END_DATA_BLOCK

DATA_BLOCK "Chan1"	// DB 21
VERSION : 0.0
BEGIN
// 392 bytes; values not shown
END_DATA_BLOCK

DATA_BLOCK "X"	// DB 31
VERSION : 0.0
BEGIN
// 140 bytes; values not shown
END_DATA_BLOCK

DATA_BLOCK "Z"	// DB 32
VERSION : 0.0
BEGIN
// 140 bytes; values not shown
END_DATA_BLOCK

DATA_BLOCK "C"	// DB 33
VERSION : 0.0
BEGIN
// 140 bytes; values not shown
END_DATA_BLOCK

DATA_BLOCK "A"	// DB 34
VERSION : 0.0
BEGIN
// 140 bytes; values not shown
END_DATA_BLOCK

DATA_BLOCK DB 77
VERSION : 0.0
BEGIN
// 88 bytes; values not shown
END_DATA_BLOCK

DATA_BLOCK "READ_DB0"	// DB 100
//KNOW_HOW_PROTECT
//
VERSION : 0.0
  STRUCT
   A1_M_NUM_ENCS_30200 : STRUCT
    SYNTAX_ID : BYTE  := B#16#82;
    bereich_u_einheit : BYTE  := B#16#61;
    spalte : WORD  := W#16#75F8;
    zeile : WORD  := W#16#1;
    bausteintyp : BYTE  := B#16#1A;
    ZEILENANZAHL : BYTE  := B#16#1;
    typ : BYTE  := B#16#3;
    laenge : BYTE  := B#16#1;
   END_STRUCT ;
   A2_M_NUM_ENCS_30200 : STRUCT
    SYNTAX_ID : BYTE  := B#16#82;
    bereich_u_einheit : BYTE  := B#16#62;
    spalte : WORD  := W#16#75F8;
    zeile : WORD  := W#16#1;
    bausteintyp : BYTE  := B#16#1A;
    ZEILENANZAHL : BYTE  := B#16#1;
    typ : BYTE  := B#16#3;
    laenge : BYTE  := B#16#1;
   END_STRUCT ;
   A3_M_NUM_ENCS_30200 : STRUCT
    SYNTAX_ID : BYTE  := B#16#82;
    bereich_u_einheit : BYTE  := B#16#63;
    spalte : WORD  := W#16#75F8;
    zeile : WORD  := W#16#1;
    bausteintyp : BYTE  := B#16#1A;
    ZEILENANZAHL : BYTE  := B#16#1;
    typ : BYTE  := B#16#3;
    laenge : BYTE  := B#16#1;
   END_STRUCT ;
   A4_M_NUM_ENCS_30200 : STRUCT
    SYNTAX_ID : BYTE  := B#16#82;
    bereich_u_einheit : BYTE  := B#16#64;
    spalte : WORD  := W#16#75F8;
    zeile : WORD  := W#16#1;
    bausteintyp : BYTE  := B#16#1A;
    ZEILENANZAHL : BYTE  := B#16#1;
    typ : BYTE  := B#16#3;
    laenge : BYTE  := B#16#1;
   END_STRUCT ;
   A5_M_NUM_ENCS_30200 : STRUCT
    SYNTAX_ID : BYTE  := B#16#82;
    bereich_u_einheit : BYTE  := B#16#65;
    spalte : WORD  := W#16#75F8;
    zeile : WORD  := W#16#1;
    bausteintyp : BYTE  := B#16#1A;
    ZEILENANZAHL : BYTE  := B#16#1;
    typ : BYTE  := B#16#3;
    laenge : BYTE  := B#16#1;
   END_STRUCT ;
   A6_M_NUM_ENCS_30200 : STRUCT
    SYNTAX_ID : BYTE  := B#16#82;
    bereich_u_einheit : BYTE  := B#16#66;
    spalte : WORD  := W#16#75F8;
    zeile : WORD  := W#16#1;
    bausteintyp : BYTE  := B#16#1A;
    ZEILENANZAHL : BYTE  := B#16#1;
    typ : BYTE  := B#16#3;
    laenge : BYTE  := B#16#1;
   END_STRUCT ;
   A7_M_NUM_ENCS_30200 : STRUCT
    SYNTAX_ID : BYTE  := B#16#82;
    bereich_u_einheit : BYTE  := B#16#67;
    spalte : WORD  := W#16#75F8;
    zeile : WORD  := W#16#1;
    bausteintyp : BYTE  := B#16#1A;
    ZEILENANZAHL : BYTE  := B#16#1;
    typ : BYTE  := B#16#3;
    laenge : BYTE  := B#16#1;
   END_STRUCT ;
   A8_M_NUM_ENCS_30200 : STRUCT
    SYNTAX_ID : BYTE  := B#16#82;
    bereich_u_einheit : BYTE  := B#16#68;
    spalte : WORD  := W#16#75F8;
    zeile : WORD  := W#16#1;
    bausteintyp : BYTE  := B#16#1A;
    ZEILENANZAHL : BYTE  := B#16#1;
    typ : BYTE  := B#16#3;
    laenge : BYTE  := B#16#1;
   END_STRUCT ;
   A21_M_LIMIT_MINUS_36100 : STRUCT
    SYNTAX_ID : BYTE  := B#16#82;
    bereich_u_einheit : BYTE  := B#16#75;
    spalte : WORD  := W#16#8D04;
    zeile : WORD  := W#16#1;
    bausteintyp : BYTE  := B#16#1A;
    ZEILENANZAHL : BYTE  := B#16#1;
    typ : BYTE  := B#16#F;
    laenge : BYTE  := B#16#8;
   END_STRUCT ;
   A21_M_LIMIT_PLUS_36110 : STRUCT
    SYNTAX_ID : BYTE  := B#16#82;
    bereich_u_einheit : BYTE  := B#16#75;
    spalte : WORD  := W#16#8D0E;
    zeile : WORD  := W#16#1;
    bausteintyp : BYTE  := B#16#1A;
    ZEILENANZAHL : BYTE  := B#16#1;
    typ : BYTE  := B#16#F;
    laenge : BYTE  := B#16#8;
   END_STRUCT ;
   A22_M_LIMIT_MINUS_36100 : STRUCT
    SYNTAX_ID : BYTE  := B#16#82;
    bereich_u_einheit : BYTE  := B#16#76;
    spalte : WORD  := W#16#8D04;
    zeile : WORD  := W#16#1;
    bausteintyp : BYTE  := B#16#1A;
    ZEILENANZAHL : BYTE  := B#16#1;
    typ : BYTE  := B#16#F;
    laenge : BYTE  := B#16#8;
   END_STRUCT ;
   A22_M_LIMIT_PLUS_36110 : STRUCT
    SYNTAX_ID : BYTE  := B#16#82;
    bereich_u_einheit : BYTE  := B#16#76;
    spalte : WORD  := W#16#8D0E;
    zeile : WORD  := W#16#1;
    bausteintyp : BYTE  := B#16#1A;
    ZEILENANZAHL : BYTE  := B#16#1;
    typ : BYTE  := B#16#F;
    laenge : BYTE  := B#16#8;
   END_STRUCT ;
   A23_M_LIMIT_MINUS_36100 : STRUCT
    SYNTAX_ID : BYTE  := B#16#82;
    bereich_u_einheit : BYTE  := B#16#77;
    spalte : WORD  := W#16#8D04;
    zeile : WORD  := W#16#1;
    bausteintyp : BYTE  := B#16#1A;
    ZEILENANZAHL : BYTE  := B#16#1;
    typ : BYTE  := B#16#F;
    laenge : BYTE  := B#16#8;
   END_STRUCT ;
   A23_M_LIMIT_PLUS_36110 : STRUCT
    SYNTAX_ID : BYTE  := B#16#82;
    bereich_u_einheit : BYTE  := B#16#77;
    spalte : WORD  := W#16#8D0E;
    zeile : WORD  := W#16#1;
    bausteintyp : BYTE  := B#16#1A;
    ZEILENANZAHL : BYTE  := B#16#1;
    typ : BYTE  := B#16#F;
    laenge : BYTE  := B#16#8;
   END_STRUCT ;
   A24_M_LIMIT_MINUS_36100 : STRUCT
    SYNTAX_ID : BYTE  := B#16#82;
    bereich_u_einheit : BYTE  := B#16#78;
    spalte : WORD  := W#16#8D04;
    zeile : WORD  := W#16#1;
    bausteintyp : BYTE  := B#16#1A;
    ZEILENANZAHL : BYTE  := B#16#1;
    typ : BYTE  := B#16#F;
    laenge : BYTE  := B#16#8;
   END_STRUCT ;
   A24_M_LIMIT_PLUS_36110 : STRUCT
    SYNTAX_ID : BYTE  := B#16#82;
    bereich_u_einheit : BYTE  := B#16#78;
    spalte : WORD  := W#16#8D0E;
    zeile : WORD  := W#16#1;
    bausteintyp : BYTE  := B#16#1A;
    ZEILENANZAHL : BYTE  := B#16#1;
    typ : BYTE  := B#16#F;
    laenge : BYTE  := B#16#8;
   END_STRUCT ;
  END_STRUCT ;	
BEGIN
   A1_M_NUM_ENCS_30200.SYNTAX_ID := B#16#82;
   A1_M_NUM_ENCS_30200.bereich_u_einheit := B#16#61;
   A1_M_NUM_ENCS_30200.spalte := W#16#75F8;
   A1_M_NUM_ENCS_30200.zeile := W#16#1;
   A1_M_NUM_ENCS_30200.bausteintyp := B#16#1A;
   A1_M_NUM_ENCS_30200.ZEILENANZAHL := B#16#1;
   A1_M_NUM_ENCS_30200.typ := B#16#3;
   A1_M_NUM_ENCS_30200.laenge := B#16#1;
   A2_M_NUM_ENCS_30200.SYNTAX_ID := B#16#82;
   A2_M_NUM_ENCS_30200.bereich_u_einheit := B#16#62;
   A2_M_NUM_ENCS_30200.spalte := W#16#75F8;
   A2_M_NUM_ENCS_30200.zeile := W#16#1;
   A2_M_NUM_ENCS_30200.bausteintyp := B#16#1A;
   A2_M_NUM_ENCS_30200.ZEILENANZAHL := B#16#1;
   A2_M_NUM_ENCS_30200.typ := B#16#3;
   A2_M_NUM_ENCS_30200.laenge := B#16#1;
   A3_M_NUM_ENCS_30200.SYNTAX_ID := B#16#82;
   A3_M_NUM_ENCS_30200.bereich_u_einheit := B#16#63;
   A3_M_NUM_ENCS_30200.spalte := W#16#75F8;
   A3_M_NUM_ENCS_30200.zeile := W#16#1;
   A3_M_NUM_ENCS_30200.bausteintyp := B#16#1A;
   A3_M_NUM_ENCS_30200.ZEILENANZAHL := B#16#1;
   A3_M_NUM_ENCS_30200.typ := B#16#3;
   A3_M_NUM_ENCS_30200.laenge := B#16#1;
   A4_M_NUM_ENCS_30200.SYNTAX_ID := B#16#82;
   A4_M_NUM_ENCS_30200.bereich_u_einheit := B#16#64;
   A4_M_NUM_ENCS_30200.spalte := W#16#75F8;
   A4_M_NUM_ENCS_30200.zeile := W#16#1;
   A4_M_NUM_ENCS_30200.bausteintyp := B#16#1A;
   A4_M_NUM_ENCS_30200.ZEILENANZAHL := B#16#1;
   A4_M_NUM_ENCS_30200.typ := B#16#3;
   A4_M_NUM_ENCS_30200.laenge := B#16#1;
   A5_M_NUM_ENCS_30200.SYNTAX_ID := B#16#82;
   A5_M_NUM_ENCS_30200.bereich_u_einheit := B#16#65;
   A5_M_NUM_ENCS_30200.spalte := W#16#75F8;
   A5_M_NUM_ENCS_30200.zeile := W#16#1;
   A5_M_NUM_ENCS_30200.bausteintyp := B#16#1A;
   A5_M_NUM_ENCS_30200.ZEILENANZAHL := B#16#1;
   A5_M_NUM_ENCS_30200.typ := B#16#3;
   A5_M_NUM_ENCS_30200.laenge := B#16#1;
   A6_M_NUM_ENCS_30200.SYNTAX_ID := B#16#82;
   A6_M_NUM_ENCS_30200.bereich_u_einheit := B#16#66;
   A6_M_NUM_ENCS_30200.spalte := W#16#75F8;
   A6_M_NUM_ENCS_30200.zeile := W#16#1;
   A6_M_NUM_ENCS_30200.bausteintyp := B#16#1A;
   A6_M_NUM_ENCS_30200.ZEILENANZAHL := B#16#1;
   A6_M_NUM_ENCS_30200.typ := B#16#3;
   A6_M_NUM_ENCS_30200.laenge := B#16#1;
   A7_M_NUM_ENCS_30200.SYNTAX_ID := B#16#82;
   A7_M_NUM_ENCS_30200.bereich_u_einheit := B#16#67;
   A7_M_NUM_ENCS_30200.spalte := W#16#75F8;
   A7_M_NUM_ENCS_30200.zeile := W#16#1;
   A7_M_NUM_ENCS_30200.bausteintyp := B#16#1A;
   A7_M_NUM_ENCS_30200.ZEILENANZAHL := B#16#1;
   A7_M_NUM_ENCS_30200.typ := B#16#3;
   A7_M_NUM_ENCS_30200.laenge := B#16#1;
   A8_M_NUM_ENCS_30200.SYNTAX_ID := B#16#82;
   A8_M_NUM_ENCS_30200.bereich_u_einheit := B#16#68;
   A8_M_NUM_ENCS_30200.spalte := W#16#75F8;
   A8_M_NUM_ENCS_30200.zeile := W#16#1;
   A8_M_NUM_ENCS_30200.bausteintyp := B#16#1A;
   A8_M_NUM_ENCS_30200.ZEILENANZAHL := B#16#1;
   A8_M_NUM_ENCS_30200.typ := B#16#3;
   A8_M_NUM_ENCS_30200.laenge := B#16#1;
   A21_M_LIMIT_MINUS_36100.SYNTAX_ID := B#16#82;
   A21_M_LIMIT_MINUS_36100.bereich_u_einheit := B#16#75;
   A21_M_LIMIT_MINUS_36100.spalte := W#16#8D04;
   A21_M_LIMIT_MINUS_36100.zeile := W#16#1;
   A21_M_LIMIT_MINUS_36100.bausteintyp := B#16#1A;
   A21_M_LIMIT_MINUS_36100.ZEILENANZAHL := B#16#1;
   A21_M_LIMIT_MINUS_36100.typ := B#16#F;
   A21_M_LIMIT_MINUS_36100.laenge := B#16#8;
   A21_M_LIMIT_PLUS_36110.SYNTAX_ID := B#16#82;
   A21_M_LIMIT_PLUS_36110.bereich_u_einheit := B#16#75;
   A21_M_LIMIT_PLUS_36110.spalte := W#16#8D0E;
   A21_M_LIMIT_PLUS_36110.zeile := W#16#1;
   A21_M_LIMIT_PLUS_36110.bausteintyp := B#16#1A;
   A21_M_LIMIT_PLUS_36110.ZEILENANZAHL := B#16#1;
   A21_M_LIMIT_PLUS_36110.typ := B#16#F;
   A21_M_LIMIT_PLUS_36110.laenge := B#16#8;
   A22_M_LIMIT_MINUS_36100.SYNTAX_ID := B#16#82;
   A22_M_LIMIT_MINUS_36100.bereich_u_einheit := B#16#76;
   A22_M_LIMIT_MINUS_36100.spalte := W#16#8D04;
   A22_M_LIMIT_MINUS_36100.zeile := W#16#1;
   A22_M_LIMIT_MINUS_36100.bausteintyp := B#16#1A;
   A22_M_LIMIT_MINUS_36100.ZEILENANZAHL := B#16#1;
   A22_M_LIMIT_MINUS_36100.typ := B#16#F;
   A22_M_LIMIT_MINUS_36100.laenge := B#16#8;
   A22_M_LIMIT_PLUS_36110.SYNTAX_ID := B#16#82;
   A22_M_LIMIT_PLUS_36110.bereich_u_einheit := B#16#76;
   A22_M_LIMIT_PLUS_36110.spalte := W#16#8D0E;
   A22_M_LIMIT_PLUS_36110.zeile := W#16#1;
   A22_M_LIMIT_PLUS_36110.bausteintyp := B#16#1A;
   A22_M_LIMIT_PLUS_36110.ZEILENANZAHL := B#16#1;
   A22_M_LIMIT_PLUS_36110.typ := B#16#F;
   A22_M_LIMIT_PLUS_36110.laenge := B#16#8;
   A23_M_LIMIT_MINUS_36100.SYNTAX_ID := B#16#82;
   A23_M_LIMIT_MINUS_36100.bereich_u_einheit := B#16#77;
   A23_M_LIMIT_MINUS_36100.spalte := W#16#8D04;
   A23_M_LIMIT_MINUS_36100.zeile := W#16#1;
   A23_M_LIMIT_MINUS_36100.bausteintyp := B#16#1A;
   A23_M_LIMIT_MINUS_36100.ZEILENANZAHL := B#16#1;
   A23_M_LIMIT_MINUS_36100.typ := B#16#F;
   A23_M_LIMIT_MINUS_36100.laenge := B#16#8;
   A23_M_LIMIT_PLUS_36110.SYNTAX_ID := B#16#82;
   A23_M_LIMIT_PLUS_36110.bereich_u_einheit := B#16#77;
   A23_M_LIMIT_PLUS_36110.spalte := W#16#8D0E;
   A23_M_LIMIT_PLUS_36110.zeile := W#16#1;
   A23_M_LIMIT_PLUS_36110.bausteintyp := B#16#1A;
   A23_M_LIMIT_PLUS_36110.ZEILENANZAHL := B#16#1;
   A23_M_LIMIT_PLUS_36110.typ := B#16#F;
   A23_M_LIMIT_PLUS_36110.laenge := B#16#8;
   A24_M_LIMIT_MINUS_36100.SYNTAX_ID := B#16#82;
   A24_M_LIMIT_MINUS_36100.bereich_u_einheit := B#16#78;
   A24_M_LIMIT_MINUS_36100.spalte := W#16#8D04;
   A24_M_LIMIT_MINUS_36100.zeile := W#16#1;
   A24_M_LIMIT_MINUS_36100.bausteintyp := B#16#1A;
   A24_M_LIMIT_MINUS_36100.ZEILENANZAHL := B#16#1;
   A24_M_LIMIT_MINUS_36100.typ := B#16#F;
   A24_M_LIMIT_MINUS_36100.laenge := B#16#8;
   A24_M_LIMIT_PLUS_36110.SYNTAX_ID := B#16#82;
   A24_M_LIMIT_PLUS_36110.bereich_u_einheit := B#16#78;
   A24_M_LIMIT_PLUS_36110.spalte := W#16#8D0E;
   A24_M_LIMIT_PLUS_36110.zeile := W#16#1;
   A24_M_LIMIT_PLUS_36110.bausteintyp := B#16#1A;
   A24_M_LIMIT_PLUS_36110.ZEILENANZAHL := B#16#1;
   A24_M_LIMIT_PLUS_36110.typ := B#16#F;
   A24_M_LIMIT_PLUS_36110.laenge := B#16#8;
END_DATA_BLOCK

DATA_BLOCK "READ_DB2"	// DB 102
VERSION : 0.0
  STRUCT
   C1_RP_rpa297_1 : STRUCT
    SYNTAX_ID : BYTE  := B#16#82;
    bereich_u_einheit : BYTE  := B#16#41;
    spalte : WORD  := W#16#1;
    zeile : WORD  := W#16#129;
    bausteintyp : BYTE  := B#16#15;
    ZEILENANZAHL : BYTE  := B#16#1;
    typ : BYTE  := B#16#F;
    laenge : BYTE  := B#16#8;
   END_STRUCT ;
   C1_RP_rpa298_1 : STRUCT
    SYNTAX_ID : BYTE  := B#16#82;
    bereich_u_einheit : BYTE  := B#16#41;
    spalte : WORD  := W#16#1;
    zeile : WORD  := W#16#12A;
    bausteintyp : BYTE  := B#16#15;
    ZEILENANZAHL : BYTE  := B#16#1;
    typ : BYTE  := B#16#F;
    laenge : BYTE  := B#16#8;
   END_STRUCT ;
   C1_RP_rpa299_1 : STRUCT
    SYNTAX_ID : BYTE  := B#16#82;
    bereich_u_einheit : BYTE  := B#16#41;
    spalte : WORD  := W#16#1;
    zeile : WORD  := W#16#12B;
    bausteintyp : BYTE  := B#16#15;
    ZEILENANZAHL : BYTE  := B#16#1;
    typ : BYTE  := B#16#F;
    laenge : BYTE  := B#16#8;
   END_STRUCT ;
   C1_RP_rpa300_1 : STRUCT
    SYNTAX_ID : BYTE  := B#16#82;
    bereich_u_einheit : BYTE  := B#16#41;
    spalte : WORD  := W#16#1;
    zeile : WORD  := W#16#12C;
    bausteintyp : BYTE  := B#16#15;
    ZEILENANZAHL : BYTE  := B#16#1;
    typ : BYTE  := B#16#F;
    laenge : BYTE  := B#16#8;
   END_STRUCT ;
   C1_RP_rpa501_1 : STRUCT
    SYNTAX_ID : BYTE  := B#16#82;
    bereich_u_einheit : BYTE  := B#16#41;
    spalte : WORD  := W#16#1;
    zeile : WORD  := W#16#1F5;
    bausteintyp : BYTE  := B#16#15;
    ZEILENANZAHL : BYTE  := B#16#1;
    typ : BYTE  := B#16#F;
    laenge : BYTE  := B#16#8;
   END_STRUCT ;
   C1_RP_rpa502_1 : STRUCT
    SYNTAX_ID : BYTE  := B#16#82;
    bereich_u_einheit : BYTE  := B#16#41;
    spalte : WORD  := W#16#1;
    zeile : WORD  := W#16#1F6;
    bausteintyp : BYTE  := B#16#15;
    ZEILENANZAHL : BYTE  := B#16#1;
    typ : BYTE  := B#16#F;
    laenge : BYTE  := B#16#8;
   END_STRUCT ;
   C1_RP_rpa503_1 : STRUCT
    SYNTAX_ID : BYTE  := B#16#82;
    bereich_u_einheit : BYTE  := B#16#41;
    spalte : WORD  := W#16#1;
    zeile : WORD  := W#16#1F7;
    bausteintyp : BYTE  := B#16#15;
    ZEILENANZAHL : BYTE  := B#16#1;
    typ : BYTE  := B#16#F;
    laenge : BYTE  := B#16#8;
   END_STRUCT ;
   C1_RP_rpa504_1 : STRUCT
    SYNTAX_ID : BYTE  := B#16#82;
    bereich_u_einheit : BYTE  := B#16#41;
    spalte : WORD  := W#16#1;
    zeile : WORD  := W#16#1F8;
    bausteintyp : BYTE  := B#16#15;
    ZEILENANZAHL : BYTE  := B#16#1;
    typ : BYTE  := B#16#F;
    laenge : BYTE  := B#16#8;
   END_STRUCT ;
  END_STRUCT ;	
BEGIN
   C1_RP_rpa297_1.SYNTAX_ID := B#16#82;
   C1_RP_rpa297_1.bereich_u_einheit := B#16#41;
   C1_RP_rpa297_1.spalte := W#16#1;
   C1_RP_rpa297_1.zeile := W#16#129;
   C1_RP_rpa297_1.bausteintyp := B#16#15;
   C1_RP_rpa297_1.ZEILENANZAHL := B#16#1;
   C1_RP_rpa297_1.typ := B#16#F;
   C1_RP_rpa297_1.laenge := B#16#8;
   C1_RP_rpa298_1.SYNTAX_ID := B#16#82;
   C1_RP_rpa298_1.bereich_u_einheit := B#16#41;
   C1_RP_rpa298_1.spalte := W#16#1;
   C1_RP_rpa298_1.zeile := W#16#12A;
   C1_RP_rpa298_1.bausteintyp := B#16#15;
   C1_RP_rpa298_1.ZEILENANZAHL := B#16#1;
   C1_RP_rpa298_1.typ := B#16#F;
   C1_RP_rpa298_1.laenge := B#16#8;
   C1_RP_rpa299_1.SYNTAX_ID := B#16#82;
   C1_RP_rpa299_1.bereich_u_einheit := B#16#41;
   C1_RP_rpa299_1.spalte := W#16#1;
   C1_RP_rpa299_1.zeile := W#16#12B;
   C1_RP_rpa299_1.bausteintyp := B#16#15;
   C1_RP_rpa299_1.ZEILENANZAHL := B#16#1;
   C1_RP_rpa299_1.typ := B#16#F;
   C1_RP_rpa299_1.laenge := B#16#8;
   C1_RP_rpa300_1.SYNTAX_ID := B#16#82;
   C1_RP_rpa300_1.bereich_u_einheit := B#16#41;
   C1_RP_rpa300_1.spalte := W#16#1;
   C1_RP_rpa300_1.zeile := W#16#12C;
   C1_RP_rpa300_1.bausteintyp := B#16#15;
   C1_RP_rpa300_1.ZEILENANZAHL := B#16#1;
   C1_RP_rpa300_1.typ := B#16#F;
   C1_RP_rpa300_1.laenge := B#16#8;
   C1_RP_rpa501_1.SYNTAX_ID := B#16#82;
   C1_RP_rpa501_1.bereich_u_einheit := B#16#41;
   C1_RP_rpa501_1.spalte := W#16#1;
   C1_RP_rpa501_1.zeile := W#16#1F5;
   C1_RP_rpa501_1.bausteintyp := B#16#15;
   C1_RP_rpa501_1.ZEILENANZAHL := B#16#1;
   C1_RP_rpa501_1.typ := B#16#F;
   C1_RP_rpa501_1.laenge := B#16#8;
   C1_RP_rpa502_1.SYNTAX_ID := B#16#82;
   C1_RP_rpa502_1.bereich_u_einheit := B#16#41;
   C1_RP_rpa502_1.spalte := W#16#1;
   C1_RP_rpa502_1.zeile := W#16#1F6;
   C1_RP_rpa502_1.bausteintyp := B#16#15;
   C1_RP_rpa502_1.ZEILENANZAHL := B#16#1;
   C1_RP_rpa502_1.typ := B#16#F;
   C1_RP_rpa502_1.laenge := B#16#8;
   C1_RP_rpa503_1.SYNTAX_ID := B#16#82;
   C1_RP_rpa503_1.bereich_u_einheit := B#16#41;
   C1_RP_rpa503_1.spalte := W#16#1;
   C1_RP_rpa503_1.zeile := W#16#1F7;
   C1_RP_rpa503_1.bausteintyp := B#16#15;
   C1_RP_rpa503_1.ZEILENANZAHL := B#16#1;
   C1_RP_rpa503_1.typ := B#16#F;
   C1_RP_rpa503_1.laenge := B#16#8;
   C1_RP_rpa504_1.SYNTAX_ID := B#16#82;
   C1_RP_rpa504_1.bereich_u_einheit := B#16#41;
   C1_RP_rpa504_1.spalte := W#16#1;
   C1_RP_rpa504_1.zeile := W#16#1F8;
   C1_RP_rpa504_1.bausteintyp := B#16#15;
   C1_RP_rpa504_1.ZEILENANZAHL := B#16#1;
   C1_RP_rpa504_1.typ := B#16#F;
   C1_RP_rpa504_1.laenge := B#16#8;
END_DATA_BLOCK

DATA_BLOCK "Program_Select"	// DB 103
//KNOW_HOW_PROTECT
//
VERSION : 0.1
  STRUCT
   program1_name : STRING  [32 ] := '_N_WORM_MPF';
   program1_path : STRING  [32 ] := '/_N_MPF_DIR/';
   program2_name : STRING  [32 ] := '_N_DRESSER_MPF';
   program2_path : STRING  [32 ] := '/_N_MPF_DIR/';
  END_STRUCT ;	
BEGIN
   program1_name := '_N_WORM_MPF';
   program1_path := '/_N_MPF_DIR/';
   program2_name := '_N_DRESSER_MPF';
   program2_path := '/_N_MPF_DIR/';
END_DATA_BLOCK

DATA_BLOCK "READ_DB3"	// DB 104
//KNOW_HOW_PROTECT
//
VERSION : 0.0
  STRUCT
   C1_RP_rpa11_R10 : STRUCT
    SYNTAX_ID : BYTE  := B#16#82;
    bereich_u_einheit : BYTE  := B#16#41;
    spalte : WORD  := W#16#1;
    zeile : WORD  := W#16#B;
    bausteintyp : BYTE  := B#16#15;
    ZEILENANZAHL : BYTE  := B#16#1;
    typ : BYTE  := B#16#F;
    laenge : BYTE  := B#16#8;
   END_STRUCT ;
   C1_RP_rpa13_R12 : STRUCT
    SYNTAX_ID : BYTE  := B#16#82;
    bereich_u_einheit : BYTE  := B#16#41;
    spalte : WORD  := W#16#1;
    zeile : WORD  := W#16#D;
    bausteintyp : BYTE  := B#16#15;
    ZEILENANZAHL : BYTE  := B#16#1;
    typ : BYTE  := B#16#F;
    laenge : BYTE  := B#16#8;
   END_STRUCT ;
   C1_RP_rpa71_R70 : STRUCT
    SYNTAX_ID : BYTE  := B#16#82;
    bereich_u_einheit : BYTE  := B#16#41;
    spalte : WORD  := W#16#1;
    zeile : WORD  := W#16#47;
    bausteintyp : BYTE  := B#16#15;
    ZEILENANZAHL : BYTE  := B#16#1;
    typ : BYTE  := B#16#F;
    laenge : BYTE  := B#16#8;
   END_STRUCT ;
   C1_RP_rpa72_R71 : STRUCT
    SYNTAX_ID : BYTE  := B#16#82;
    bereich_u_einheit : BYTE  := B#16#41;
    spalte : WORD  := W#16#1;
    zeile : WORD  := W#16#48;
    bausteintyp : BYTE  := B#16#15;
    ZEILENANZAHL : BYTE  := B#16#1;
    typ : BYTE  := B#16#F;
    laenge : BYTE  := B#16#8;
   END_STRUCT ;
   C1_RP_rpa73_R72 : STRUCT
    SYNTAX_ID : BYTE  := B#16#82;
    bereich_u_einheit : BYTE  := B#16#41;
    spalte : WORD  := W#16#1;
    zeile : WORD  := W#16#49;
    bausteintyp : BYTE  := B#16#15;
    ZEILENANZAHL : BYTE  := B#16#1;
    typ : BYTE  := B#16#F;
    laenge : BYTE  := B#16#8;
   END_STRUCT ;
   C1_RP_rpa74_R73 : STRUCT
    SYNTAX_ID : BYTE  := B#16#82;
    bereich_u_einheit : BYTE  := B#16#41;
    spalte : WORD  := W#16#1;
    zeile : WORD  := W#16#4A;
    bausteintyp : BYTE  := B#16#15;
    ZEILENANZAHL : BYTE  := B#16#1;
    typ : BYTE  := B#16#F;
    laenge : BYTE  := B#16#8;
   END_STRUCT ;
   C1_RP_rpa501_R500 : STRUCT
    SYNTAX_ID : BYTE  := B#16#82;
    bereich_u_einheit : BYTE  := B#16#41;
    spalte : WORD  := W#16#1;
    zeile : WORD  := W#16#1F5;
    bausteintyp : BYTE  := B#16#15;
    ZEILENANZAHL : BYTE  := B#16#1;
    typ : BYTE  := B#16#F;
    laenge : BYTE  := B#16#8;
   END_STRUCT ;
   C1_RP_rpa502_R501 : STRUCT
    SYNTAX_ID : BYTE  := B#16#82;
    bereich_u_einheit : BYTE  := B#16#41;
    spalte : WORD  := W#16#1;
    zeile : WORD  := W#16#1F6;
    bausteintyp : BYTE  := B#16#15;
    ZEILENANZAHL : BYTE  := B#16#1;
    typ : BYTE  := B#16#F;
    laenge : BYTE  := B#16#8;
   END_STRUCT ;
   C1_RP_rpa503_R502 : STRUCT
    SYNTAX_ID : BYTE  := B#16#82;
    bereich_u_einheit : BYTE  := B#16#41;
    spalte : WORD  := W#16#1;
    zeile : WORD  := W#16#1F7;
    bausteintyp : BYTE  := B#16#15;
    ZEILENANZAHL : BYTE  := B#16#1;
    typ : BYTE  := B#16#F;
    laenge : BYTE  := B#16#8;
   END_STRUCT ;
   C1_RP_rpa504_R503 : STRUCT
    SYNTAX_ID : BYTE  := B#16#82;
    bereich_u_einheit : BYTE  := B#16#41;
    spalte : WORD  := W#16#1;
    zeile : WORD  := W#16#1F8;
    bausteintyp : BYTE  := B#16#15;
    ZEILENANZAHL : BYTE  := B#16#1;
    typ : BYTE  := B#16#F;
    laenge : BYTE  := B#16#8;
   END_STRUCT ;
   C1_RP_rpa505_R504 : STRUCT
    SYNTAX_ID : BYTE  := B#16#82;
    bereich_u_einheit : BYTE  := B#16#41;
    spalte : WORD  := W#16#1;
    zeile : WORD  := W#16#1F9;
    bausteintyp : BYTE  := B#16#15;
    ZEILENANZAHL : BYTE  := B#16#1;
    typ : BYTE  := B#16#F;
    laenge : BYTE  := B#16#8;
   END_STRUCT ;
   C1_RP_rpa506_R505 : STRUCT
    SYNTAX_ID : BYTE  := B#16#82;
    bereich_u_einheit : BYTE  := B#16#41;
    spalte : WORD  := W#16#1;
    zeile : WORD  := W#16#1FA;
    bausteintyp : BYTE  := B#16#15;
    ZEILENANZAHL : BYTE  := B#16#1;
    typ : BYTE  := B#16#F;
    laenge : BYTE  := B#16#8;
   END_STRUCT ;
   C1_RP_rpa507_R506 : STRUCT
    SYNTAX_ID : BYTE  := B#16#82;
    bereich_u_einheit : BYTE  := B#16#41;
    spalte : WORD  := W#16#1;
    zeile : WORD  := W#16#1FB;
    bausteintyp : BYTE  := B#16#15;
    ZEILENANZAHL : BYTE  := B#16#1;
    typ : BYTE  := B#16#F;
    laenge : BYTE  := B#16#8;
   END_STRUCT ;
   C1_RP_rpa508_R507 : STRUCT
    SYNTAX_ID : BYTE  := B#16#82;
    bereich_u_einheit : BYTE  := B#16#41;
    spalte : WORD  := W#16#1;
    zeile : WORD  := W#16#1FC;
    bausteintyp : BYTE  := B#16#15;
    ZEILENANZAHL : BYTE  := B#16#1;
    typ : BYTE  := B#16#F;
    laenge : BYTE  := B#16#8;
   END_STRUCT ;
   C1_RP_rpa509_R508 : STRUCT
    SYNTAX_ID : BYTE  := B#16#82;
    bereich_u_einheit : BYTE  := B#16#41;
    spalte : WORD  := W#16#1;
    zeile : WORD  := W#16#1FD;
    bausteintyp : BYTE  := B#16#15;
    ZEILENANZAHL : BYTE  := B#16#1;
    typ : BYTE  := B#16#F;
    laenge : BYTE  := B#16#8;
   END_STRUCT ;
   C1_RP_rpa510_R509 : STRUCT
    SYNTAX_ID : BYTE  := B#16#82;
    bereich_u_einheit : BYTE  := B#16#41;
    spalte : WORD  := W#16#1;
    zeile : WORD  := W#16#1FE;
    bausteintyp : BYTE  := B#16#15;
    ZEILENANZAHL : BYTE  := B#16#1;
    typ : BYTE  := B#16#F;
    laenge : BYTE  := B#16#8;
   END_STRUCT ;
  END_STRUCT ;	
BEGIN
   C1_RP_rpa11_R10.SYNTAX_ID := B#16#82;
   C1_RP_rpa11_R10.bereich_u_einheit := B#16#41;
   C1_RP_rpa11_R10.spalte := W#16#1;
   C1_RP_rpa11_R10.zeile := W#16#B;
   C1_RP_rpa11_R10.bausteintyp := B#16#15;
   C1_RP_rpa11_R10.ZEILENANZAHL := B#16#1;
   C1_RP_rpa11_R10.typ := B#16#F;
   C1_RP_rpa11_R10.laenge := B#16#8;
   C1_RP_rpa13_R12.SYNTAX_ID := B#16#82;
   C1_RP_rpa13_R12.bereich_u_einheit := B#16#41;
   C1_RP_rpa13_R12.spalte := W#16#1;
   C1_RP_rpa13_R12.zeile := W#16#D;
   C1_RP_rpa13_R12.bausteintyp := B#16#15;
   C1_RP_rpa13_R12.ZEILENANZAHL := B#16#1;
   C1_RP_rpa13_R12.typ := B#16#F;
   C1_RP_rpa13_R12.laenge := B#16#8;
   C1_RP_rpa71_R70.SYNTAX_ID := B#16#82;
   C1_RP_rpa71_R70.bereich_u_einheit := B#16#41;
   C1_RP_rpa71_R70.spalte := W#16#1;
   C1_RP_rpa71_R70.zeile := W#16#47;
   C1_RP_rpa71_R70.bausteintyp := B#16#15;
   C1_RP_rpa71_R70.ZEILENANZAHL := B#16#1;
   C1_RP_rpa71_R70.typ := B#16#F;
   C1_RP_rpa71_R70.laenge := B#16#8;
   C1_RP_rpa72_R71.SYNTAX_ID := B#16#82;
   C1_RP_rpa72_R71.bereich_u_einheit := B#16#41;
   C1_RP_rpa72_R71.spalte := W#16#1;
   C1_RP_rpa72_R71.zeile := W#16#48;
   C1_RP_rpa72_R71.bausteintyp := B#16#15;
   C1_RP_rpa72_R71.ZEILENANZAHL := B#16#1;
   C1_RP_rpa72_R71.typ := B#16#F;
   C1_RP_rpa72_R71.laenge := B#16#8;
   C1_RP_rpa73_R72.SYNTAX_ID := B#16#82;
   C1_RP_rpa73_R72.bereich_u_einheit := B#16#41;
   C1_RP_rpa73_R72.spalte := W#16#1;
   C1_RP_rpa73_R72.zeile := W#16#49;
   C1_RP_rpa73_R72.bausteintyp := B#16#15;
   C1_RP_rpa73_R72.ZEILENANZAHL := B#16#1;
   C1_RP_rpa73_R72.typ := B#16#F;
   C1_RP_rpa73_R72.laenge := B#16#8;
   C1_RP_rpa74_R73.SYNTAX_ID := B#16#82;
   C1_RP_rpa74_R73.bereich_u_einheit := B#16#41;
   C1_RP_rpa74_R73.spalte := W#16#1;
   C1_RP_rpa74_R73.zeile := W#16#4A;
   C1_RP_rpa74_R73.bausteintyp := B#16#15;
   C1_RP_rpa74_R73.ZEILENANZAHL := B#16#1;
   C1_RP_rpa74_R73.typ := B#16#F;
   C1_RP_rpa74_R73.laenge := B#16#8;
   C1_RP_rpa501_R500.SYNTAX_ID := B#16#82;
   C1_RP_rpa501_R500.bereich_u_einheit := B#16#41;
   C1_RP_rpa501_R500.spalte := W#16#1;
   C1_RP_rpa501_R500.zeile := W#16#1F5;
   C1_RP_rpa501_R500.bausteintyp := B#16#15;
   C1_RP_rpa501_R500.ZEILENANZAHL := B#16#1;
   C1_RP_rpa501_R500.typ := B#16#F;
   C1_RP_rpa501_R500.laenge := B#16#8;
   C1_RP_rpa502_R501.SYNTAX_ID := B#16#82;
   C1_RP_rpa502_R501.bereich_u_einheit := B#16#41;
   C1_RP_rpa502_R501.spalte := W#16#1;
   C1_RP_rpa502_R501.zeile := W#16#1F6;
   C1_RP_rpa502_R501.bausteintyp := B#16#15;
   C1_RP_rpa502_R501.ZEILENANZAHL := B#16#1;
   C1_RP_rpa502_R501.typ := B#16#F;
   C1_RP_rpa502_R501.laenge := B#16#8;
   C1_RP_rpa503_R502.SYNTAX_ID := B#16#82;
   C1_RP_rpa503_R502.bereich_u_einheit := B#16#41;
   C1_RP_rpa503_R502.spalte := W#16#1;
   C1_RP_rpa503_R502.zeile := W#16#1F7;
   C1_RP_rpa503_R502.bausteintyp := B#16#15;
   C1_RP_rpa503_R502.ZEILENANZAHL := B#16#1;
   C1_RP_rpa503_R502.typ := B#16#F;
   C1_RP_rpa503_R502.laenge := B#16#8;
   C1_RP_rpa504_R503.SYNTAX_ID := B#16#82;
   C1_RP_rpa504_R503.bereich_u_einheit := B#16#41;
   C1_RP_rpa504_R503.spalte := W#16#1;
   C1_RP_rpa504_R503.zeile := W#16#1F8;
   C1_RP_rpa504_R503.bausteintyp := B#16#15;
   C1_RP_rpa504_R503.ZEILENANZAHL := B#16#1;
   C1_RP_rpa504_R503.typ := B#16#F;
   C1_RP_rpa504_R503.laenge := B#16#8;
   C1_RP_rpa505_R504.SYNTAX_ID := B#16#82;
   C1_RP_rpa505_R504.bereich_u_einheit := B#16#41;
   C1_RP_rpa505_R504.spalte := W#16#1;
   C1_RP_rpa505_R504.zeile := W#16#1F9;
   C1_RP_rpa505_R504.bausteintyp := B#16#15;
   C1_RP_rpa505_R504.ZEILENANZAHL := B#16#1;
   C1_RP_rpa505_R504.typ := B#16#F;
   C1_RP_rpa505_R504.laenge := B#16#8;
   C1_RP_rpa506_R505.SYNTAX_ID := B#16#82;
   C1_RP_rpa506_R505.bereich_u_einheit := B#16#41;
   C1_RP_rpa506_R505.spalte := W#16#1;
   C1_RP_rpa506_R505.zeile := W#16#1FA;
   C1_RP_rpa506_R505.bausteintyp := B#16#15;
   C1_RP_rpa506_R505.ZEILENANZAHL := B#16#1;
   C1_RP_rpa506_R505.typ := B#16#F;
   C1_RP_rpa506_R505.laenge := B#16#8;
   C1_RP_rpa507_R506.SYNTAX_ID := B#16#82;
   C1_RP_rpa507_R506.bereich_u_einheit := B#16#41;
   C1_RP_rpa507_R506.spalte := W#16#1;
   C1_RP_rpa507_R506.zeile := W#16#1FB;
   C1_RP_rpa507_R506.bausteintyp := B#16#15;
   C1_RP_rpa507_R506.ZEILENANZAHL := B#16#1;
   C1_RP_rpa507_R506.typ := B#16#F;
   C1_RP_rpa507_R506.laenge := B#16#8;
   C1_RP_rpa508_R507.SYNTAX_ID := B#16#82;
   C1_RP_rpa508_R507.bereich_u_einheit := B#16#41;
   C1_RP_rpa508_R507.spalte := W#16#1;
   C1_RP_rpa508_R507.zeile := W#16#1FC;
   C1_RP_rpa508_R507.bausteintyp := B#16#15;
   C1_RP_rpa508_R507.ZEILENANZAHL := B#16#1;
   C1_RP_rpa508_R507.typ := B#16#F;
   C1_RP_rpa508_R507.laenge := B#16#8;
   C1_RP_rpa509_R508.SYNTAX_ID := B#16#82;
   C1_RP_rpa509_R508.bereich_u_einheit := B#16#41;
   C1_RP_rpa509_R508.spalte := W#16#1;
   C1_RP_rpa509_R508.zeile := W#16#1FD;
   C1_RP_rpa509_R508.bausteintyp := B#16#15;
   C1_RP_rpa509_R508.ZEILENANZAHL := B#16#1;
   C1_RP_rpa509_R508.typ := B#16#F;
   C1_RP_rpa509_R508.laenge := B#16#8;
   C1_RP_rpa510_R509.SYNTAX_ID := B#16#82;
   C1_RP_rpa510_R509.bereich_u_einheit := B#16#41;
   C1_RP_rpa510_R509.spalte := W#16#1;
   C1_RP_rpa510_R509.zeile := W#16#1FE;
   C1_RP_rpa510_R509.bausteintyp := B#16#15;
   C1_RP_rpa510_R509.ZEILENANZAHL := B#16#1;
   C1_RP_rpa510_R509.typ := B#16#F;
   C1_RP_rpa510_R509.laenge := B#16#8;
END_DATA_BLOCK

DATA_BLOCK "X_BACK"	// DB 106
//KNOW_HOW_PROTECT
//
VERSION : 0.1
  STRUCT
   program1_name : STRING  [32 ] := '_N_ASUP1_SPF';
   program1_path : STRING  [32 ] := '/_N_CMA_DIR/';
   program2_name : STRING  [32 ] := '_N_ASUP2_SPF';
   program2_path : STRING  [32 ] := '/_N_CMA_DIR/';
  END_STRUCT ;	
BEGIN
   program1_name := '_N_ASUP1_SPF';
   program1_path := '/_N_CMA_DIR/';
   program2_name := '_N_ASUP2_SPF';
   program2_path := '/_N_CMA_DIR/';
END_DATA_BLOCK

// DB 110: know-how protected block, not included

DATA_BLOCK "USER_DB0"	// DB 120
VERSION : 0.0
  STRUCT
   STAT0 : ARRAY  [0 .. 100 ] OF WORD ;
  END_STRUCT ;	
BEGIN
   STAT0[0] := W#16#102;
   STAT0[1] := W#16#201;
   STAT0[2] := W#16#101;
   STAT0[3] := W#16#101;
   STAT0[5] := W#16#46E2;
   STAT0[6] := W#16#9000;
   STAT0[10] := W#16#4516;
   STAT0[15] := W#16#453B;
   STAT0[16] := W#16#8000;
   STAT0[20] := W#16#4CBE;
   STAT0[21] := W#16#BC20;
   STAT0[25] := W#16#4CBE;
   STAT0[26] := W#16#BC20;
   STAT0[30] := W#16#CCBE;
   STAT0[31] := W#16#BC20;
   STAT0[35] := W#16#CCBE;
   STAT0[36] := W#16#BC20;
   STAT0[40] := W#16#CCBE;
   STAT0[41] := W#16#BC20;
   STAT0[45] := W#16#CCBE;
   STAT0[46] := W#16#BC20;
   STAT0[47] := W#16#71;
   STAT0[48] := W#16#4800;
   STAT0[55] := W#16#C294;
   STAT0[56] := W#16#E353;
   STAT0[60] := W#16#4320;
END_DATA_BLOCK

DATA_BLOCK "USER_DB1"	// DB 121
VERSION : 0.0
  STRUCT
   STAT0 : ARRAY  [0 .. 100 ] OF WORD ;
  END_STRUCT ;	
BEGIN
   STAT0[0] := W#16#102;
   STAT0[1] := W#16#201;
   STAT0[2] := W#16#101;
   STAT0[3] := W#16#101;
   STAT0[5] := W#16#46E2;
   STAT0[6] := W#16#9000;
   STAT0[10] := W#16#4516;
   STAT0[15] := W#16#453B;
   STAT0[16] := W#16#8000;
   STAT0[20] := W#16#4CBE;
   STAT0[21] := W#16#BC20;
   STAT0[25] := W#16#4CBE;
   STAT0[26] := W#16#BC20;
   STAT0[30] := W#16#CCBE;
   STAT0[31] := W#16#BC20;
   STAT0[35] := W#16#CCBE;
   STAT0[36] := W#16#BC20;
   STAT0[40] := W#16#CCBE;
   STAT0[41] := W#16#BC20;
   STAT0[45] := W#16#CCBE;
   STAT0[46] := W#16#BC20;
   STAT0[47] := W#16#71;
   STAT0[48] := W#16#4800;
   STAT0[55] := W#16#C294;
   STAT0[56] := W#16#E353;
   STAT0[60] := W#16#4320;
END_DATA_BLOCK

DATA_BLOCK "USER_DB2"	// DB 122
VERSION : 0.0
  STRUCT
   STAT0 : ARRAY  [0 .. 100 ] OF WORD ;
  END_STRUCT ;	
BEGIN
   STAT0[0] := W#16#45E1;
   STAT0[1] := W#16#A37B;
   STAT0[45] := W#16#7148;
   STAT0[47] := W#16#71;
   STAT0[48] := W#16#4800;
   STAT0[50] := W#16#3E8;
   STAT0[55] := W#16#47C3;
   STAT0[56] := W#16#5000;
END_DATA_BLOCK

DATA_BLOCK "USER_DB3"	// DB 123
VERSION : 0.0
  STRUCT
   STAT0 : ARRAY  [0 .. 100 ] OF WORD ;
  END_STRUCT ;	
BEGIN
   STAT0[0] := W#16#45E1;
   STAT0[1] := W#16#A37B;
   STAT0[45] := W#16#7148;
   STAT0[47] := W#16#71;
   STAT0[48] := W#16#4800;
   STAT0[50] := W#16#3E8;
   STAT0[55] := W#16#47C3;
   STAT0[56] := W#16#5000;
END_DATA_BLOCK

DATA_BLOCK "USER_DB4"	// DB 124
VERSION : 0.0
  STRUCT
   STAT0 : ARRAY  [0 .. 100 ] OF WORD ;
  END_STRUCT ;	
BEGIN
   STAT0[0] := W#16#45E1;
   STAT0[1] := W#16#A37B;
   STAT0[45] := W#16#7148;
   STAT0[47] := W#16#71;
   STAT0[48] := W#16#4800;
   STAT0[50] := W#16#3E8;
   STAT0[55] := W#16#47C3;
   STAT0[56] := W#16#5000;
END_DATA_BLOCK

DATA_BLOCK "USER_DB5"	// DB 125
VERSION : 0.0
  STRUCT
   STAT0 : ARRAY  [0 .. 100 ] OF WORD ;
  END_STRUCT ;	
BEGIN
   STAT0[0] := W#16#45E1;
   STAT0[1] := W#16#A37B;
   STAT0[45] := W#16#7148;
   STAT0[47] := W#16#71;
   STAT0[48] := W#16#4800;
   STAT0[50] := W#16#3E8;
   STAT0[55] := W#16#47C3;
   STAT0[56] := W#16#5000;
END_DATA_BLOCK

DATA_BLOCK "USER_DB6"	// DB 126
VERSION : 0.1
  STRUCT
   STAT0 : ARRAY  [0 .. 100 ] OF WORD ;
  END_STRUCT ;	
BEGIN
END_DATA_BLOCK

DATA_BLOCK "USER_DB7"	// DB 127
VERSION : 0.1
  STRUCT
   STAT0 : ARRAY  [0 .. 100 ] OF
   WORD ;
  END_STRUCT ;	
BEGIN
END_DATA_BLOCK

DATA_BLOCK "USER_DB8"	// DB 128
VERSION : 0.1
  STRUCT
   STAT0 : ARRAY  [0 .. 100 ] OF WORD ;
  END_STRUCT ;	
BEGIN
END_DATA_BLOCK

DATA_BLOCK "USER_DB9"	// DB 129
VERSION : 0.1
  STRUCT
   STAT0 : ARRAY  [0 .. 100 ] OF WORD ;
  END_STRUCT ;	
BEGIN
END_DATA_BLOCK

DATA_BLOCK DB 150
AUTHOR : NUMERIK
FAMILY : _800D
VERSION : 0.0
"GET"
BEGIN
END_DATA_BLOCK

DATA_BLOCK DB 151
AUTHOR : NUMERIK
FAMILY : _800D
VERSION : 0.0
"GET"
BEGIN
END_DATA_BLOCK

DATA_BLOCK DB 153
AUTHOR : NUMERIK
FAMILY : _800D
VERSION : 0.0
"GET"
BEGIN
END_DATA_BLOCK

DATA_BLOCK DB 154
AUTHOR : NUMERIK
FAMILY : _800D
VERSION : 0.0
"GET"
BEGIN
END_DATA_BLOCK

DATA_BLOCK DB 155
AUTHOR : NUMERIK
FAMILY : _800D
VERSION : 0.0
"GET"
BEGIN
END_DATA_BLOCK

DATA_BLOCK DB 156
AUTHOR : NUMERIK
FAMILY : _800D
VERSION : 0.0
"PUT"
BEGIN
END_DATA_BLOCK

DATA_BLOCK DB 157
AUTHOR : NUMERIK
FAMILY : _800D
VERSION : 0.0
"PI_SERV"
BEGIN
END_DATA_BLOCK

DATA_BLOCK DB 158
AUTHOR : NUMERIK
FAMILY : _800D
VERSION : 0.0
"PI_SERV"
BEGIN
END_DATA_BLOCK

DATA_BLOCK DB 159
AUTHOR : NUMERIK
FAMILY : _800D
VERSION : 0.0
"PI_SERV"
BEGIN
END_DATA_BLOCK

DATA_BLOCK DB 160
AUTHOR : NUMERIK
FAMILY : _800D
VERSION : 0.0
"PI_SERV"
BEGIN
END_DATA_BLOCK

DATA_BLOCK "CtrlE"	// DB 1000
TITLE = Datainterface Ctrl-Energy
AUTHOR : NUMERIK
FAMILY : _800D
NAME : CTRL_E
VERSION : 4.5
  STRUCT
   Profile : ARRAY  [1 .. 8 ] OF STRUCT
    ESaveOn : BOOL ;	// Activate energy-saving profile immediately
    ReloadT2 : BOOL ;	// Reload Prewarning time (T2)
    res0_2 : BOOL ;
    res0_3 : BOOL ;
    res0_4 : BOOL ;
    res0_5 : BOOL ;
    res0_6 : BOOL ;
    res0_7 : BOOL ;
    HmiESaveOn : BOOL ;	// HMI->PLC: Activate energy-saving profile immediately
    res1_1 : BOOL ;
    res1_2 : BOOL ;
    res1_3 : BOOL ;
    res1_4 : BOOL ;
    res1_5 : BOOL ;
    res1_6 : BOOL ;
    res1_7 : BOOL ;
    MasterCompSig : BOOL ;	// Master computer signal
    PlcUserSig : BOOL ;	// PLC user signal
    res2_2 : BOOL ;
    res2_3 : BOOL ;
    res2_4 : BOOL ;
    res2_5 : BOOL ;
    res2_6 : BOOL ;
    res2_7 : BOOL ;
    res3 : BYTE ;
    ESaveIsOn : BOOL ;	// Energy-saving state active
    T1Expired : BOOL ;	// Activation time T1 expired
    res4_2 : BOOL ;
    res4_3 : BOOL ;
    res4_4 : BOOL ;
    res4_5 : BOOL ;
    res4_6 : BOOL ;
    res4_7 : BOOL ;
    res5 : BYTE ;
    ActValT1 : INT ;	// T1 current value
    ActValT2 : INT ;	// T2 current value
    ESaveValid : BOOL ;	// HMI->PLC: Energy-saving profile valid
    ESaveOff : BOOL ;	// HMI->PLC: Deactivate energy-saving profileblock energy-saving profile
    res10_2 : BOOL ;
    res10_3 : BOOL ;
    res10_4 : BOOL ;
    res10_5 : BOOL ;
    res10_6 : BOOL ;
    res10_7 : BOOL ;
    CondOpPanel : BOOL ;	// HMI->PLC: Operator panel
    CondDataTransfer : BOOL ;	// HMI->PLC: Data transfer
    CondWindowChange : BOOL ;	// HMI->PLC: Window change
    res11_3 : BOOL ;
    res11_4 : BOOL ;
    res11_5 : BOOL ;
    res11_6 : BOOL ;
    res11_7 : BOOL ;
    CondMCP : BOOL ;	// HMI->PLC: Machine control panel
    res12_1 : BOOL ;
    res12_2 : BOOL ;
    res12_3 : BOOL ;
    res12_4 : BOOL ;
    res12_5 : BOOL ;
    res12_6 : BOOL ;
    res12_7 : BOOL ;
    CondNcChan1 : BOOL ;	// HMI->PLC: NC channel 1 in reset
    CondNcChan2 : BOOL ;	// HMI->PLC: NC channel 2 in reset
    CondNcChan3 : BOOL ;	// HMI->PLC: NC channel 3 in reset
    CondNcChan4 : BOOL ;	// HMI->PLC: NC channel 4 in reset
    CondNcChan5 : BOOL ;	// HMI->PLC: NC channel 5 in reset
    CondNcChan6 : BOOL ;	// HMI->PLC: NC channel 6 in reset
    CondNcChan7 : BOOL ;	// HMI->PLC: NC channel 7 in reset
    CondNcChan8 : BOOL ;	// HMI->PLC: NC channel 8 in reset
    CondNcChan9 : BOOL ;	// HMI->PLC: NC channel 9 in reset
    CondNcChan10 : BOOL ;	// HMI->PLC: NC channel 10 in reset
    res14_2 : BOOL ;
    res14_3 : BOOL ;
    res14_4 : BOOL ;
    res14_5 : BOOL ;
    res14_6 : BOOL ;
    res14_7 : BOOL ;
    CondMasterCompSig : BOOL ;	// HMI->PLC: Master computer signal
    CondPlcUserSig : BOOL ;	// HMI->PLC: PLC user signal
    res15_2 : BOOL ;
    res15_3 : BOOL ;
    res15_4 : BOOL ;
    res15_5 : BOOL ;
    res15_6 : BOOL ;
    res15_7 : BOOL ;
    PresetT1 : INT ;	// HMI->PLC: Activation time T1
    PresetT2 : INT ;	// HMI->PLC: Prewarning time T2
   END_STRUCT ;
  END_STRUCT ;	
BEGIN
   Profile[1].ESaveValid := TRUE;
   Profile[1].ESaveOff := TRUE;
   Profile[1].CondNcChan1 := TRUE;
   Profile[1].CondNcChan2 := TRUE;
   Profile[1].CondNcChan3 := TRUE;
   Profile[1].CondNcChan4 := TRUE;
   Profile[1].CondNcChan5 := TRUE;
   Profile[1].CondNcChan6 := TRUE;
   Profile[1].CondNcChan7 := TRUE;
   Profile[1].CondNcChan8 := TRUE;
   Profile[1].CondNcChan9 := TRUE;
   Profile[1].CondNcChan10 := TRUE;
   Profile[1].CondPlcUserSig := TRUE;
   Profile[1].PresetT1 := 60;
   Profile[1].PresetT2 := 120;
   Profile[2].ESaveValid := TRUE;
   Profile[2].ESaveOff := TRUE;
   Profile[2].CondMCP := TRUE;
   Profile[2].CondNcChan1 := TRUE;
   Profile[2].CondNcChan2 := TRUE;
   Profile[2].CondNcChan3 := TRUE;
   Profile[2].CondNcChan4 := TRUE;
   Profile[2].CondNcChan5 := TRUE;
   Profile[2].CondNcChan6 := TRUE;
   Profile[2].CondNcChan7 := TRUE;
   Profile[2].CondNcChan8 := TRUE;
   Profile[2].CondNcChan9 := TRUE;
   Profile[2].CondNcChan10 := TRUE;
   Profile[2].CondPlcUserSig := TRUE;
   Profile[2].PresetT1 := 120;
   Profile[2].PresetT2 := 300;
   Profile[3].ESaveValid := TRUE;
   Profile[3].ESaveOff := TRUE;
   Profile[3].CondOpPanel := TRUE;
   Profile[3].CondDataTransfer := TRUE;
   Profile[3].CondWindowChange := TRUE;
   Profile[3].CondMCP := TRUE;
   Profile[3].CondNcChan1 := TRUE;
   Profile[3].CondNcChan2 := TRUE;
   Profile[3].CondNcChan3 := TRUE;
   Profile[3].CondNcChan4 := TRUE;
   Profile[3].CondNcChan5 := TRUE;
   Profile[3].CondNcChan6 := TRUE;
   Profile[3].CondNcChan7 := TRUE;
   Profile[3].CondNcChan8 := TRUE;
   Profile[3].CondNcChan9 := TRUE;
   Profile[3].CondNcChan10 := TRUE;
   Profile[3].CondPlcUserSig := TRUE;
   Profile[3].PresetT1 := 600;
END_DATA_BLOCK

DATA_BLOCK "SentronPac"	// DB 1001
TITLE = Datainterface SentronPac
AUTHOR : NUMERIK
FAMILY : _800D
NAME : SENTRONP
VERSION : 4.5
  STRUCT
   ManualVal : BOOL ;	// Display of manual value
   SentronPacMach : BOOL ;	// Sentron PAC represented machine
   FeedInEnergyReadSP : BOOL ;	// Feed in energy read from Sentron PAC
   FeedBackEnergyReadSP : BOOL ;	// Feed back energy read from Sentron PAC
   res0_4 : BOOL ;	// reserved
   res0_5 : BOOL ;	// reserved
   res0_6 : BOOL ;	// reserved
   res0_7 : BOOL ;	// reserved
   MeasAuto : BOOL ;	// measurement by PLC basic programm
   res1_1 : BOOL ;	// reserved
   res1_2 : BOOL ;	// reserved
   res1_3 : BOOL ;	// reserved
   res1_4 : BOOL ;	// reserved
   res1_5 : BOOL ;	// reserved
   res1_6 : BOOL ;	// reserved
   res1_7 : BOOL ;	// reserved
   MeasAct : BOOL ;	// Active measurement
   res3 : BYTE ;	// reserved
   ManualValue : REAL ;	// Manual value
   ActivePowerItem : REAL ;	// Active power item
   ActiveEnergyItem : REAL ;	// Active energy item
   ReactiveEnergyItem : REAL ;	// Reactive energy item
   ActivePowerSentron : REAL ;	// Active power from Sentron
   ActiveEnergySentron : REAL ;	// Active energy  from Sentron
   ReactiveEnergySentron : REAL ;	// Reactive energy  from Sentron
   ActiveEnergyDay : REAL ;	// Active energy day
   ReactiveEnergyDay : REAL ;	// Reactive energy day
   ActiveEnergyPrevDay : REAL ;	// Active energy previous day
   ReactiveEnergyPrevDay : REAL ;	// Reactive energy  previous day
   ActiveEnergyMonth : REAL ;	// Active energy month
   ReactiveEnergyMonth : REAL ;	// Reactive energy month
   ActiveEnergyPrevMonth : REAL ;	// Active energy previous month
   ReactiveEnergyPrevMonth : REAL ;	// Reactive energy previous month
   ActiveEnergyYear : REAL ;	// Active energy year
   ReactiveEnergyYear : REAL ;	// Reactive energy year
   ActiveEnergyPrevYear : REAL ;	// Active energy previous year
   ReactiveEnergyPrevYear : REAL ;	// Reactive energy previous year
   res80 : BYTE ;	// reserved
   res81 : BYTE ;	// reserved
   res82 : BYTE ;	// reserved
   res83 : BYTE ;	// reserved
   res84 : BYTE ;	// reserved
   res85 : BYTE ;	// reserved
   res86 : BYTE ;	// reserved
   res87 : BYTE ;	// reserved
   res88 : REAL ;	// reserved
   res92 : REAL ;	// reserved
  END_STRUCT ;	
BEGIN
END_DATA_BLOCK

ORGANIZATION_BLOCK OB 1
VERSION : 1.0
VAR_TEMP
  OB1_EV_CLASS : BYTE ;
  OB1_SCAN_1 : BYTE ;
  OB1_PRIORITY : BYTE ;
  OB1_OB_NUMBR : BYTE ;
  OB1_RESERVED_1 : BYTE ;
  OB1_RESERVED_2 : BYTE ;
  OB1_PREV_CYCLE : INT ;
  OB1_MIN_CYCLE : INT ;
  OB1_MAX_CYCLE : INT ;
  OB1_DATE_TIME : DATE_AND_TIME ;
END_VAR
BEGIN
NETWORK
TITLE = Reset
      CALL  "GP_HP";
      CALL  "MCP_IFM" (
           $1                       := B#16#1,
           $2                       := B#16#1,
           $3                       := B#16#3,
           $4                       := DB2.DBX 185.6,
           $5                       := P#M 500.0);
      CALL  "AL_MSG" (
           $1                       := TRUE,
           $2                       := "Reset_Key");
      A     "Reset_Key";
      =     DB21.DBX 7.7;
      AN    DB11.DBX 7.2;
      =     DB21.DBX 6.6;
      =     DB21.DBX 6.7;
      A     "Refpoint_Key";
      =     DB21.DBX 1.0;
      CALL  "Functions block call";
      BE;
END_ORGANIZATION_BLOCK

ORGANIZATION_BLOCK OB 40
VERSION : 1.0
VAR_TEMP
  OB40_EV_CLASS : BYTE ;
  OB40_STRT_INF : BYTE ;
  OB40_PRIORITY : BYTE ;
  OB40_OB_NUMBR : BYTE ;
  OB40_RESERVED_1 : BYTE ;
  OB40_MDL_ID : BYTE ;
  OB40_MDL_ADDR : INT ;
  OB40_POINT_ADDR : DWORD ;
  OB40_DATE_TIME : DATE_AND_TIME ;	//data for the Basic program
  GP_IRFromNCK : BOOL ;	//Interrupt from NCK
  GP_TM : BOOL ;	//Toolmanagment
  GP_InPosition : ARRAY  [1 .. 31 ] OF BOOL ;	//InPos Signal from FC15,16,18
  GP_AuxFunction : ARRAY  [1 .. 10 ] OF BOOL ;	//auxiliary functions
  GP_FMBlock : ARRAY  [1 .. 10 ] OF BOOL ;	//not used
//Insert User-data from here
END_VAR
BEGIN
NETWORK
TITLE =
      CALL  "GP_PRAL";
//Insert User program from here
END_ORGANIZATION_BLOCK

